# B&R Automation Studio project Panasonic_LinkaPowerCP2_A2021055 (part 24)

#### Main.st - Init, cyclic, exit code
```iecst
PROGRAM _INIT

END_PROGRAM

PROGRAM _CYCLIC

	//Volanie funkcie SequenceControl//
	SequenceControl(SC:= SC_P2_Cistenie);

	//Volanie podprogramov//
	OvlDveri;

	//Reset sekcie //
	IF P2_Cistenie.Reset THEN
		SC_P2_Cistenie.Step:= 0;
		P2_Cistenie.Reset:= FALSE;
	ELSIF NOT Safety.STAV.Linka_ZonaCS_AKTIVNA THEN
		SC_P2_Cistenie.Step:= 0;
	END_IF

	CASE SC_P2_Cistenie.Step OF

		0:
			SC_P2_Cistenie.StepName:='0 - Nulovanie';
			SC_OvlDveri.Step:= 0;
			P2_Cistenie.Automat:= FALSE;
			P2_Cistenie.KoniecCyklu:= FALSE;
			P2_Cistenie.Manual:= FALSE;
			P2_Cistenie.STAV.PoINIT:= FALSE;
			P2_Cistenie.OUT.Ionizator_OFF:= TRUE;
			P2_Cistenie.OUT.OdsavanieOfuk_ON:= FALSE;
			P2_Cistenie.OUT.Odsavanie_ON:= FALSE;
			P2_Cistenie.OUT.VzduchPreIonizator_ON:= FALSE;
			P2_Robot.COM_OUT.Cistenie_BezpecnaPozicia:= FALSE;
			P2_Robot.COM_OUT.Cistenie_OdoberPowerCP_4F:= FALSE;
			P2_Robot.COM_OUT.Cistenie_OdoberPowerCP_5F:= FALSE;
			P2_Robot.COM_OUT.Cistenie_OdoberPowerCP_5H:= FALSE;
			P2_Robot.COM_OUT.Cistenie_OtacajPowerCP:= FALSE;
			P2_Robot.COM_OUT.Cistenie_PolozPowerCP_4F:= FALSE;
			P2_Robot.COM_OUT.Cistenie_PolozPowerCP_5F:= FALSE;
			P2_Robot.COM_OUT.Cistenie_PolozPowerCP_5H:= FALSE;

			P2_Cistenie.COM_OUT.Stav_CistenieUkoncene:= FALSE;

			IF Safety.STAV.Linka_ZonaCS_AKTIVNA AND
				Safety.STAV.P2_ZonaBunky_AKTIVNA AND
				P2_Pracovisko.STAV.HardwareBunky_OK AND
				NOT P2_Pracovisko.STAV.Porucha_ST2 AND
				NOT P2_Pracovisko.STAV.Porucha_ST3 AND
				NOT P2_Pracovisko.STAV.Porucha_ST4 AND
				NOT P2_Pracovisko.STAV.Porucha_ST5 THEN
				SC_P2_Cistenie.ResetStep:= TRUE;
				SC_P2_Cistenie.Step:= 1;
			END_IF

		1:
			SC_P2_Cistenie.StepName:='1 - Cakam na spustenie vyroby';
			P2_Cistenie.KoniecCyklu:= FALSE;
			IF P2_Cistenie.Automat THEN
				SC_P2_Cistenie.Step:= 2;
			ELSIF P2_Cistenie.Manual THEN
				SC_P2_Cistenie.Step:= 700;
			END_IF

			//********************************************************Inicializácia****************************************************************************//

		2:
			SC_P2_Cistenie.StepName:='2 - Inicializacia - cakam na spustenie inicializacie';
			SC_P2_Cistenie.IdleTime.PT:= T#500ms;
			SC_P2_Cistenie.AlarmTime.PT:= T#5s;
			SC_P2_Cistenie.IdleTime.IN:= TRUE;

			IF SC_P2_Cistenie.IdleTime.Q THEN
				SC_P2_Cistenie.ResetStep:= TRUE;
				SC_P2_Cistenie.Step:= 3;
			END_IF

		3:
			SC_P2_Cistenie.StepName:='2 - Inicializacia - otvorenie dveri';
			SC_P2_Cistenie.IdleTime.PT:= T#500ms;
			SC_P2_Cistenie.AlarmTime.PT:= T#5s;

			IF NOT SC_P2_Cistenie.Switch1 THEN
				Dvere_OTVOR:= TRUE;
				SC_P2_Cistenie.Switch1:= TRUE;
			END_IF

			IF P2_Cistenie.IN.Dvere_OTVORENE THEN
				P2_Robot.COM_OUT.Cistenie_BezpecnaPozicia:= TRUE;
				P2_Cistenie.STAV.PoINIT:= TRUE;
				SC_P2_Cistenie.ResetStep:= TRUE;
				SC_P2_Cistenie.Step:= 100;
			END_IF

			//********************************************************Automatický režim****************************************************************************//

		100:
			SC_P2_Cistenie.StepName:='100 - Automaticky Rezim - cakam na spustenie cistenia';
			SC_P2_Cistenie.IdleTime.PT:= T#200ms;
			SC_P2_Cistenie.AlarmTime.PT:= T#5s;

			IF P2_Cistenie.KoniecCyklu AND NOT P2_StoperZvarania.Automat THEN
				SC_P2_Cistenie.ResetStep:= TRUE;
				SC_P2_Cistenie.Step:= 0;
			ELSIF P2_Cistenie.COM_IN.Cistenie_START THEN
				SC_P2_Cistenie.ResetStep:= TRUE;
				SC_P2_Cistenie.Step:= 102;
			END_IF

		102:
			SC_P2_Cistenie.StepName:='102 - Automaticky Rezim - vystavenie signalu pre robota odober Power CP z paletky a presun do cistenia';
			SC_P2_Cistenie.IdleTime.PT:= T#200ms;
			SC_P2_Cistenie.AlarmTime.PT:= T#5s;

			IF NOT P2_Robot.COM_IN.Stav_Cistenie_PowerCP_v_Cisteni AND NOT P2_Cistenie.IN.Vakum_OK THEN
				P2_Robot.COM_OUT.Cistenie_BezpecnaPozicia:= TRUE;
				IF Linka.PAR.ZvolenyModel = '4F' THEN
					P2_Robot.COM_OUT.Cistenie_OdoberPowerCP_4F:= TRUE;
					P2_Cistenie.OUT.Odsavanie_ON:= TRUE;
					SC_P2_Cistenie.ResetStep:= TRUE;
					SC_P2_Cistenie.Step:= 105;
				ELSIF Linka.PAR.ZvolenyModel = '5F' THEN
					P2_Robot.COM_OUT.Cistenie_OdoberPowerCP_5F:= TRUE;
					P2_Cistenie.OUT.Odsavanie_ON:= TRUE;
					SC_P2_Cistenie.ResetStep:= TRUE;
					SC_P2_Cistenie.Step:= 105;
				ELSIF Linka.PAR.ZvolenyModel = '5H' THEN
					P2_Robot.COM_OUT.Cistenie_OdoberPowerCP_5H:= TRUE;
					P2_Cistenie.OUT.Odsavanie_ON:= TRUE;
					SC_P2_Cistenie.ResetStep:= TRUE;
					SC_P2_Cistenie.Step:= 105;
				END_IF
			END_IF

		105:
			SC_P2_Cistenie.StepName:='105 - Automaticky Rezim - cakam na signal robot odobral Power CP z paletky';
			SC_P2_Cistenie.IdleTime.PT:= T#200ms;
			SC_P2_Cistenie.AlarmTime.PT:= T#5s;

			IF P2_Robot.COM_IN.Stav_Cistenie_PowerCP_v_Cisteni THEN
				P2_Robot.COM_OUT.Cistenie_OdoberPowerCP_4F:= FALSE;
				P2_Robot.COM_OUT.Cistenie_OdoberPowerCP_5F:= FALSE;
				P2_Robot.COM_OUT.Cistenie_OdoberPowerCP_5H:= FALSE;
				SC_P2_Cistenie.ResetStep:= TRUE;
				SC_P2_Cistenie.Step:= 108;
			END_IF

		108:
			SC_P2_Cistenie.StepName:='108 - Automaticky Rezim - zatvorenie dveri, spustenie ionizatora';
			SC_P2_Cistenie.IdleTime.PT:= T#2s;
			SC_P2_Cistenie.AlarmTime.PT:= T#5s;

			IF NOT SC_P2_Cistenie.Switch1 THEN
				P2_Cistenie.OUT.Ionizator_OFF:= FALSE;
				P2_Cistenie.OUT.VzduchPreIonizator_ON:= TRUE;
				Dvere_ZATVOR:= TRUE;
				P2_Robot.COM_OUT.Cistenie_BezpecnaPozicia:= FALSE;
				SC_P2_Cistenie.Switch1:= TRUE;
			END_IF

			IF P2_Cistenie.IN.Dvere_ZATVORENE THEN
				SC_P2_Cistenie.ResetStep:= TRUE;
				SC_P2_Cistenie.Step:= 112;
			END_IF

		112:
			SC_P2_Cistenie.StepName:='112 - Automaticky Rezim - zapnutie ofuku';
			SC_P2_Cistenie.IdleTime.PT:= T#2s;
			SC_P2_Cistenie.AlarmTime.PT:= T#5s;

			IF P2_Cistenie.IN.Vakum_OK THEN
				P2_Cistenie.OUT.OdsavanieOfuk_ON:= TRUE;
				SC_P2_Cistenie.ResetStep:= TRUE;
				SC_P2_Cistenie.Step:= 115;
			END_IF

		115:
			SC_P2_Cistenie.StepName:='115 - Automaticky Rezim - vystavenie signalu pre robota vykonaj otacanie Power CP v cisteni';
			SC_P2_Cistenie.IdleTime.PT:= T#200ms;
			SC_P2_Cistenie.AlarmTime.PT:= T#5s;

			IF NOT P2_Robot.COM_IN.Stav_Cistenie_Otacanie_Ukoncene THEN
				P2_Robot.COM_OUT.Cistenie_OtacajPowerCP:= TRUE;
				SC_P2_Cistenie.ResetStep:= TRUE;
				SC_P2_Cistenie.Step:= 118;
			END_IF

		118:
			SC_P2_Cistenie.StepName:='118 - Automaticky Rezim - cakam na signal robot ukoncil otacanie Power CP';
			SC_P2_Cistenie.IdleTime.PT:= T#200ms;
			SC_P2_Cistenie.AlarmTime.PT:= T#5s;

			IF P2_Robot.COM_IN.Stav_Cistenie_Otacanie_Ukoncene THEN
				P2_Robot.COM_OUT.Cistenie_OtacajPowerCP:= FALSE;
				SC_P2_Cistenie.ResetStep:= TRUE;
				SC_P2_Cistenie.Step:= 120;
			END_IF

		120:
			SC_P2_Cistenie.StepName:='120 - Automaticky Rezim - otvorenie dveri,vypnutie ofuku a odsavania';
			SC_P2_Cistenie.IdleTime.PT:= T#2s;
			SC_P2_Cistenie.AlarmTime.PT:= T#5s;

			IF NOT SC_P2_Cistenie.Switch1 THEN
				P2_Cistenie.OUT.OdsavanieOfuk_ON:= FALSE;
				P2_Cistenie.OUT.Odsavanie_ON:= FALSE;
				Dvere_OTVOR:= TRUE;
				SC_P2_Cistenie.Switch1:= TRUE;
			END_IF

			IF P2_Cistenie.IN.Dvere_OTVORENE THEN
				P2_Cistenie.OUT.Ionizator_OFF:= TRUE;
				P2_Cistenie.OUT.VzduchPreIonizator_ON:= FALSE;
				P2_Robot.COM_OUT.Cistenie_BezpecnaPozicia:= TRUE;
				SC_P2_Cistenie.ResetStep:= TRUE;
				SC_P2_Cistenie.Step:= 122;
			END_IF

		122:
			SC_P2_Cistenie.StepName:='122 - Automaticky Rezim - vystavenie signalu pre robota poloz Power CP na paletku po cisteni';
			SC_P2_Cistenie.IdleTime.PT:= T#200ms;
			SC_P2_Cistenie.AlarmTime.PT:= T#5s;

			IF NOT P2_Robot.COM_IN.Stav_Cistenie_PowerCP_Polozene THEN
				IF Linka.PAR.ZvolenyModel = '4F' THEN
					P2_Robot.COM_OUT.Cistenie_PolozPowerCP_4F:= TRUE;
					SC_P2_Cistenie.ResetStep:= TRUE;
					SC_P2_Cistenie.Step:= 125;
				ELSIF Linka.PAR.ZvolenyModel = '5F' THEN
					P2_Robot.COM_OUT.Cistenie_PolozPowerCP_5F:= TRUE;
					SC_P2_Cistenie.ResetStep:= TRUE;
					SC_P2_Cistenie.Step:= 125;
				ELSIF Linka.PAR.ZvolenyModel = '5H' THEN
					P2_Robot.COM_OUT.Cistenie_PolozPowerCP_5H:= TRUE;
					SC_P2_Cistenie.ResetStep:= TRUE;
					SC_P2_Cistenie.Step:= 125;
				END_IF
			END_IF

		125:
			SC_P2_Cistenie.StepName:='125 - Automaticky Rezim - cakam na signal robot polozil Power CP na paletku';
			SC_P2_Cistenie.IdleTime.PT:= T#200ms;
			SC_P2_Cistenie.AlarmTime.PT:= T#5s;

			IF P2_Robot.COM_IN.Stav_Cistenie_PowerCP_Polozene THEN
				P2_Robot.COM_OUT.Cistenie_PolozPowerCP_4F:= FALSE;
				P2_Robot.COM_OUT.Cistenie_PolozPowerCP_5F:= FALSE;
				P2_Robot.COM_OUT.Cistenie_PolozPowerCP_5H:= FALSE;
				SC_P2_Cistenie.ResetStep:= TRUE;
				SC_P2_Cistenie.Step:= 128;
			END_IF

		128:
			SC_P2_Cistenie.StepName:='122 - Automaticky Rezim - vystavenie signalu ukoncenie cistenia';
			SC_P2_Cistenie.IdleTime.PT:= T#200ms;
			SC_P2_Cistenie.AlarmTime.PT:= T#5s;

			IF NOT SC_P2_Cistenie.Switch1 THEN
				P2_Cistenie.COM_OUT.Stav_CistenieUkoncene:= TRUE;
				SC_P2_Cistenie.Switch1:= TRUE;
			END_IF

			IF NOT P2_Cistenie.COM_IN.Cistenie_START THEN
				P2_Cistenie.COM_OUT.Stav_CistenieUkoncene:= FALSE;
				SC_P2_Cistenie.ResetStep:= TRUE;
				SC_P2_Cistenie.Step:= 100;
			END_IF

			//**************************************************Ručný režim***********************************************************//

		700:
			SC_P2_Cistenie.StepName:='700 - Rucny rezim';
			SC_P2_Cistenie.IdleTime.PT:= T#200ms;
			SC_P2_Cistenie.AlarmTime.PT:= T#5s;

			//Otvorenie zatvorenie čistenia//
			IF P2_Cistenie.CMD.RR_Cistenie_OTVOR THEN
				Dvere_OTVOR:= TRUE;
				P2_Cistenie.CMD.RR_Cistenie_OTVOR:= FALSE;
			ELSIF P2_Cistenie.CMD.RR_Cistenie_ZATVOR THEN
				Dvere_ZATVOR:= TRUE;
				P2_Cistenie.CMD.RR_Cistenie_ZATVOR:= FALSE;
			END_IF

	END_CASE

END_PROGRAM

PROGRAM _EXIT
	(* Insert code here *)

END_PROGRAM
```

#### Variables.var - Local variables
```iecst
VAR
	SC_OvlDveri : SequenceControlTyp;
	Dvere_OTVOR : BOOL;
	Dvere_ZATVOR : BOOL;
END_VAR
```

#### OvlDveri.st
```iecst
ACTION OvlDveri:

	//Volanie funkcie SequenceControl//
	SequenceControl(SC:= SC_OvlDveri);

	CASE SC_OvlDveri.Step OF

		0:
			SC_OvlDveri.StepName:= '0 - Nulovanie';
			Dvere_OTVOR:= FALSE;
			Dvere_ZATVOR:= FALSE;
			P2_Cistenie.OUT.Dvere_OTVOR:= FALSE;
			P2_Cistenie.OUT.Dvere_ZATVOR:= FALSE;

			IF SC_P2_Cistenie.Step <> 0 THEN
				SC_OvlDveri.ResetStep:= TRUE;
				SC_OvlDveri.Step:= 1;
			END_IF

		1:
			SC_OvlDveri.StepName:= '1 - Rozhodnutie o cinnosti';
			IF Dvere_OTVOR THEN
				SC_OvlDveri.Step:= 10;
			ELSIF Dvere_ZATVOR THEN
				SC_OvlDveri.Step:= 20;
			END_IF

		10:
			SC_OvlDveri.StepName:= '10 - Otvorenie dveri';
			SC_OvlDveri.IdleTime.PT:= T#3s;
			SC_OvlDveri.AlarmTime.PT:= T#3s;

			IF P2_Cistenie.Automat THEN
				SC_OvlDveri.AlarmTime.IN:= TRUE;
			ELSE
				SC_OvlDveri.IdleTime.IN:= TRUE;
			END_IF

			IF NOT SC_OvlDveri.Switch1 THEN
				P2_Cistenie.OUT.Dvere_OTVOR:= TRUE;
				SC_OvlDveri.Switch1:= TRUE;
			END_IF

			IF P2_Cistenie.IN.Dvere_OTVORENE OR SC_OvlDveri.IdleTime.Q THEN
				SC_OvlDveri.ResetStep:= TRUE;
				SC_OvlDveri.Step:= 0;
			ELSIF SC_OvlDveri.AlarmTime.Q THEN
				P2_Alarmy[224]:= TRUE;
				P2_Pracovisko.STAV.Porucha_ST5:= TRUE;
			END_IF

		20:
			SC_OvlDveri.StepName:= '20 - Zatvorenie dveri';
			SC_OvlDveri.IdleTime.PT:= T#3s;
			SC_OvlDveri.AlarmTime.PT:= T#3s;

			IF P2_Cistenie.Automat THEN
				SC_OvlDveri.AlarmTime.IN:= TRUE;
			ELSE
				SC_OvlDveri.IdleTime.IN:= TRUE;
			END_IF

			IF NOT SC_OvlDveri.Switch1 THEN
				P2_Cistenie.OUT.Dvere_ZATVOR:= TRUE;
				SC_OvlDveri.Switch1:= TRUE;
			END_IF

			IF P2_Cistenie.IN.Dvere_ZATVORENE OR SC_OvlDveri.IdleTime.Q THEN
				SC_OvlDveri.ResetStep:= TRUE;
				SC_OvlDveri.Step:= 0;
			ELSIF SC_OvlDveri.AlarmTime.Q THEN
				P2_Alarmy[223]:= TRUE;
				P2_Pracovisko.STAV.Porucha_ST5:= TRUE;
			END_IF

	END_CASE

END_ACTION
```

### Program Logical/Program/Pracovisko_2/P2_OvladVizu (IEC)

#### Main.st - Init, cyclic, exit code
```iecst
PROGRAM _INIT
	(* Insert code here *)

END_PROGRAM

PROGRAM _CYCLIC

	//*************************************Prepnutie obrazovky pri stlačení tlačítka CS*********************************//
	IF EDGEPOS(P2_Pracovisko.STAV.Manual AND NOT Safety.STAV.Linka_ZonaCS_AKTIVNA) THEN
		P2_Vizu.GoPage:= 'PageAutomatP2';
	END_IF

	//************************************Filter alarmov**************************************************************//
	FilterVizu_P2:= '[{"logicalOperator":"and","value":200,"conditionType":">=","columnType":"cod","useAlarmState":false,"alarmState":0},{"value":299,"conditionType":"<=","columnType":"cod","useAlarmState":false,"alarmState":0}]';

	//**********************************Zobrazenie upozornenia na kontrolu skrutiek na stanici 5 skrutkovania***********************************//
	IF EDGEPOS(Linka.PAR.ZvolenyModel = '4F')THEN
		P2_Vizu.ZobrazHL5_ST5:= TRUE;
		P2_Vizu.ZobrazHL6_ST5:= FALSE;
		P2_Vizu.ZobrazHL7_ST5:= FALSE;
	END_IF

	IF EDGEPOS(Linka.PAR.ZvolenyModel = '5F')THEN
		P2_Vizu.ZobrazHL5_ST5:= FALSE;
		P2_Vizu.ZobrazHL6_ST5:= TRUE;
		P2_Vizu.ZobrazHL7_ST5:= FALSE;
	END_IF

	IF EDGEPOS(Linka.PAR.ZvolenyModel = '5H')THEN
		P2_Vizu.ZobrazHL5_ST5:= FALSE;
		P2_Vizu.ZobrazHL6_ST5:= FALSE;
		P2_Vizu.ZobrazHL7_ST5:= TRUE;
	END_IF

	//Zmeny farieb tlačítok ovládania zámkov//
	//Zadné dvere //
	IF P2_Pracovisko.STAV.ZadneDvereZamknute AND P2_Pracovisko.IN.ZadneDvereLS_PritomnostAdaptera AND P2_Pracovisko.IN.ZadneDverePS_PritomnostAdaptera THEN
		P2_Vizu.TL_ZadnyZamok_Farba:= "Button_Green";
	ELSIF P2_Pracovisko.IN.ZadneDvereLS_PritomnostAdaptera AND P2_Pracovisko.IN.ZadneDverePS_PritomnostAdaptera THEN
		IF Blikac1s THEN
			P2_Vizu.TL_ZadnyZamok_Farba:= "Button_Blue";
		ELSE
			P2_Vizu.TL_ZadnyZamok_Farba:= "Operate";
		END_IF
	ELSE
		P2_Vizu.TL_ZadnyZamok_Farba:= "Button_Red";
	END_IF

	//Predné dvere //
	IF P2_Pracovisko.STAV.PredneDvereZamknute AND P2_Pracovisko.IN.PredneDvereLS_PritomnostAdaptera AND P2_Pracovisko.IN.PredneDverePS_PritomnostAdaptera THEN
		P2_Vizu.TL_PrednyZamok_Farba:= "Button_Green";
	ELSIF P2_Pracovisko.IN.PredneDvereLS_PritomnostAdaptera AND P2_Pracovisko.IN.PredneDverePS_PritomnostAdaptera THEN
		IF Blikac1s THEN
			P2_Vizu.TL_PrednyZamok_Farba:= "Button_Blue";
		ELSE
			P2_Vizu.TL_PrednyZamok_Farba:= "Operate";
		END_IF
	ELSE
		P2_Vizu.TL_PrednyZamok_Farba:= "Button_Red";
	END_IF

	//***********************************Zobrazenie warningov pracoviska****************************************************//
	//0 - Pracovisko je vypnuté.
	//1 - Prebieha inicializácia pracoviska.
	//2 - Na pracovisku prebieha výroba.
	//3 - Prebieha ukončenie pracovného cyklu pracoviska.
	//4 - Prebieha režim vyprázdnenia linky.
	//5 - Robot nie je prepnuty do automatického režimu !!!
	//6 - Doplň zásobník matíc M4 !!!
	//7 - Doplň zásobník skrutiek M4 !!!
	//8 - Doplň zásobník skrutiek M5 !!!
	//9 - Doplň zásobník skrutiek M6 !!!

	IF NOT P2_Robot.COM_IN.Stav_RezimAUTOMAT THEN
		P2_Vizu.Warnings_Index:= 5;
	ELSIF P2_Pracovisko.STAV.Automat AND NOT P2_Pracovisko.STAV.PoINIT AND NOT P2_Pracovisko.STAV.UkoncenieCyklu_BUSY THEN
		P2_Vizu.Warnings_Index:= 1;
	ELSIF P2_StoperMaticovacky.SkrutSet_MaticaM4.IN.ZasobnikMaticPrazdny THEN
		P2_Vizu.Warnings_Index:= 6;
	ELSIF P2_Srobovanie.SkrutSet_M4.IN.ZasobnikSkrutiekPrazdny THEN
		P2_Vizu.Warnings_Index:= 7;
	ELSIF P2_Srobovanie.SkrutSet_M5.IN.VibracnyHrniec.PritomnostSkrutiekVHrnci THEN
		P2_Vizu.Warnings_Index:= 8;
	ELSIF P2_Srobovanie.SkrutSet_M6.IN.VibracnyHrniec.PritomnostSkrutiekVHrnci THEN
		P2_Vizu.Warnings_Index:= 9;
	ELSIF Linka.PAR.TestovaciKus THEN
		P2_Vizu.Warnings_Index:= 11;
	ELSIF Linka.PAR.VyprazdnenieLinky THEN
		P2_Vizu.Warnings_Index:= 4;
	ELSIF P2_Pracovisko.STAV.PoINIT AND NOT P2_Pracovisko.STAV.UkoncenieCyklu_BUSY THEN
		P2_Vizu.Warnings_Index:= 2;
	ELSIF P2_Pracovisko.STAV.UkoncenieCyklu_BUSY THEN
		P2_Vizu.Warnings_Index:= 3;
	ELSIF NOT P2_Pracovisko.STAV.Automat THEN
		P2_Vizu.Warnings_Index:= 0;
	END_IF

	//************************Prepínanie farby textového pola warning zariadenia***********************************//
	IF P2_Vizu.Warnings_Index = 0 THEN
		P2_Vizu.Warnings_Farba:= "TextOutput_Grey";
	ELSIF P2_Vizu.Warnings_Index = 1 THEN
		P2_Vizu.Warnings_Farba:= "TextOutput_Blue";
	ELSIF P2_Vizu.Warnings_Index = 2 THEN
		P2_Vizu.Warnings_Farba:= "TextOutput_Green";
	ELSIF P2_Vizu.Warnings_Index = 3 THEN
		P2_Vizu.Warnings_Farba:= "TextOutput_Blue";
	ELSIF P2_Vizu.Warnings_Index = 4 THEN
		P2_Vizu.Warnings_Farba:= "TextOutput_Green";
	ELSIF P2_Vizu.Warnings_Index = 11 THEN
		P2_Vizu.Warnings_Farba:= "TextOutput_Green";
	ELSE
		IF Blikac1s THEN
			P2_Vizu.Warnings_Farba:= "TextOutput_Orange";
		ELSE
			P2_Vizu.Warnings_Farba:= "TextOutput_Grey";
		END_IF
	END_IF

	//***********************Prepnutie bootovacej obrazovky********************************//
	IF P2_Vizu.ActualPage <> 'PageBootP2' AND NOT Safety.STAV.Linka_SafetyPLC_Nabehlo THEN
		P2_Vizu.GoPage:= 'PageBootP2';
	ELSIF P2_Vizu.ActualPage = 'PageBootP2' AND Safety.STAV.Linka_SafetyPLC_Nabehlo THEN
		P2_Vizu.GoPage:= 'PageAutomatP2';
	END_IF

	IF P2_Vizu.GoPage = 'PageBootP2' AND P2_Vizu.ActualPage = 'PageBootP2' THEN
		P2_Vizu.GoPage:= '';
	ELSIF P2_Vizu.GoPage = 'PageAutomatP2' AND P2_Vizu.ActualPage = 'PageAutomatP2' THEN
		P2_Vizu.GoPage:= '';
	END_IF

	//********************************Blikanie tlačítka Alarmy*******************************************************//
	IF P2_Pracovisko.STAV.PORUCHA AND P2_Vizu.ActualPage <> 'PageAlarmP2' THEN
		IF Blikac500ms THEN
			P2_AlarmyVizu.FarbaTlacitka_Alarmy:= "Button_Red";
		ELSE
			P2_AlarmyVizu.FarbaTlacitka_Alarmy:= "default";
		END_IF
	ELSE
		P2_AlarmyVizu.FarbaTlacitka_Alarmy:= "default";
	END_IF

	//*************************************Zamknutie tlačítok***************************************************************//
	//Zamknutie tlačítok ovládania zámkov//
	IF P2_Pracovisko.STAV.Automat THEN
		P2_Vizu.TL_OvladaniaZamkov_ENABLE:= FALSE;
	ELSIF P2_Srobovanie.STAV.RR_Polohovanie_BUSY THEN
		P2_Vizu.TL_OvladaniaZamkov_ENABLE:= FALSE;
	ELSIF P2_Srobovanie.STAV.CistenieSkrutkovackyM5_BUSY THEN
		P2_Vizu.TL_OvladaniaZamkov_ENABLE:= FALSE;
	ELSIF P2_Srobovanie.STAV.CistenieSkrutkovackyM6_BUSY THEN
		P2_Vizu.TL_OvladaniaZamkov_ENABLE:= FALSE;
	ELSIF P2_Zvaranie.STAV.RR_SekvenciaZvarania_BUSY THEN
		P2_Vizu.TL_OvladaniaZamkov_ENABLE:= FALSE;
	ELSE
		P2_Vizu.TL_OvladaniaZamkov_ENABLE:= TRUE;
	END_IF

	//Tlačítko Štat Automat//
	IF P2_Pracovisko.STAV.UkoncenieCyklu_BUSY THEN
		P2_Vizu.TL_StartAutomat_ENABLE:= FALSE;
	ELSIF P2_Pracovisko.STAV.PORUCHA THEN
		P2_Vizu.TL_StartAutomat_ENABLE:= FALSE;
	ELSIF NOT P2_Robot.COM_IN.Stav_RezimAUTOMAT THEN
		P2_Vizu.TL_StartAutomat_ENABLE:= FALSE;
	ELSIF NOT Safety.STAV.P2_ZonaBunky_AKTIVNA THEN
		P2_Vizu.TL_StartAutomat_ENABLE:= FALSE;
	ELSIF NOT P2_Pracovisko.STAV.HardwareZaklTesnenia_OK THEN
		P2_Vizu.TL_StartAutomat_ENABLE:= FALSE;
	ELSIF NOT P2_Pracovisko.STAV.HardwareBunky_OK THEN
		P2_Vizu.TL_StartAutomat_ENABLE:= FALSE;
	ELSE
		P2_Vizu.TL_StartAutomat_ENABLE:= TRUE;
	END_IF

	//Tlačítko Ukončenie Cyklu//
	IF P2_Pracovisko.STAV.PoINIT THEN
		P2_Vizu.TL_KoniecCyklu_ENABLE:= TRUE;
	ELSE
		P2_Vizu.TL_KoniecCyklu_ENABLE:= FALSE;
	END_IF

	//Tlačítko STOP//
	IF P2_Pracovisko.STAV.PoINIT AND NOT P2_Pracovisko.STAV.UkoncenieCyklu_BUSY THEN
		P2_Vizu.TL_STOP_ENABLE:= FALSE;
	ELSE
		P2_Vizu.TL_STOP_ENABLE:= TRUE;
	END_IF

	//Tlačítko Režim Automat//
	P2_Vizu.TL_RezimAutomat_ENABLE:= TRUE;

	//Tlačítko Režim Manual//
	IF P2_Pracovisko.STAV.Automat THEN
		P2_Vizu.TL_RezimManual_ENABLE:= FALSE;
	ELSIF NOT P2_Pracovisko.STAV.HardwareZaklTesnenia_OK THEN
		P2_Vizu.TL_RezimManual_ENABLE:= FALSE;
	ELSIF NOT P2_Pracovisko.STAV.HardwareBunky_OK THEN
		P2_Vizu.TL_RezimManual_ENABLE:= FALSE;
	ELSE
		P2_Vizu.TL_RezimManual_ENABLE:= TRUE;
	END_IF

	//RR - Tlačítko vysunutia maticovačky//
	IF NOT Safety.STAV.P2_ZonaBunky_AKTIVNA THEN
		P2_Vizu.TL_VysunutiaMaticovacM4_ENABLE:= FALSE;
	ELSE
		P2_Vizu.TL_VysunutiaMaticovacM4_ENABLE:= TRUE;
	END_IF

	//RR - Tlačítko čistenia skrutkovačky M6//
	IF P2_Srobovanie.STAV.RR_Polohovanie_BUSY THEN
		P2_Vizu.TL_VycistiSkrutkovackuM6_ENABLE:= FALSE;
	ELSIF NOT Safety.STAV.P2_ZonaBunky_AKTIVNA THEN
		P2_Vizu.TL_VycistiSkrutkovackuM6_ENABLE:= FALSE;
	ELSIF NOT Safety.STAV.Linka_ZonaCS_AKTIVNA THEN
		P2_Vizu.TL_VycistiSkrutkovackuM6_ENABLE:= FALSE;
	ELSIF P2_Srobovanie.STAV.CistenieSkrutkovackyM6_BUSY THEN
		P2_Vizu.TL_VycistiSkrutkovackuM6_ENABLE:= FALSE;
	ELSIF P2_Srobovanie.STAV.CistenieSkrutkovackyM5_BUSY THEN
		P2_Vizu.TL_VycistiSkrutkovackuM6_ENABLE:= FALSE;
	ELSIF NOT P2_Pracovisko.STAV.SkrutkovackyZasunute THEN
		P2_Vizu.TL_VycistiSkrutkovackuM6_ENABLE:= FALSE;
	ELSIF P2_Srobovanie.CMD.RR_SkrutSetM6_VysunBrzdu THEN
		P2_Vizu.TL_VycistiSkrutkovackuM6_ENABLE:= FALSE;
	ELSIF P2_Srobovanie.CMD.RR_SkrutSetM6_Zasobnik_RUN THEN
		P2_Vizu.TL_VycistiSkrutkovackuM6_ENABLE:= FALSE;
	ELSE
		P2_Vizu.TL_VycistiSkrutkovackuM6_ENABLE:= TRUE;
	END_IF

	//RR - Tlačítko čistenia skrutkovačky M5//
	IF P2_Srobovanie.STAV.RR_Polohovanie_BUSY THEN
		P2_Vizu.TL_VycistiSkrutkovackuM5_ENABLE:= FALSE;
	ELSIF NOT Safety.STAV.P2_ZonaBunky_AKTIVNA THEN
		P2_Vizu.TL_VycistiSkrutkovackuM5_ENABLE:= FALSE;
	ELSIF NOT Safety.STAV.Linka_ZonaCS_AKTIVNA THEN
		P2_Vizu.TL_VycistiSkrutkovackuM5_ENABLE:= FALSE;
	ELSIF P2_Srobovanie.STAV.CistenieSkrutkovackyM6_BUSY THEN
		P2_Vizu.TL_VycistiSkrutkovackuM5_ENABLE:= FALSE;
	ELSIF P2_Srobovanie.STAV.CistenieSkrutkovackyM5_BUSY THEN
		P2_Vizu.TL_VycistiSkrutkovackuM5_ENABLE:= FALSE;
	ELSIF NOT P2_Pracovisko.STAV.SkrutkovackyZasunute THEN
		P2_Vizu.TL_VycistiSkrutkovackuM5_ENABLE:= FALSE;
	ELSIF P2_Srobovanie.CMD.RR_SkrutSetM5_VysunBrzdu THEN
		P2_Vizu.TL_VycistiSkrutkovackuM5_ENABLE:= FALSE;
	ELSIF P2_Srobovanie.CMD.RR_SkrutSetM5_Zasobnik_RUN THEN
		P2_Vizu.TL_VycistiSkrutkovackuM5_ENABLE:= FALSE;
	ELSE
		P2_Vizu.TL_VycistiSkrutkovackuM5_ENABLE:= TRUE;
	END_IF

	//RR - Tlačítko polohovania aplikátora//
	IF P2_Srobovanie.STAV.RR_Polohovanie_BUSY THEN
		P2_Vizu.TL_PolohujManipulator_ENABLE:= FALSE;
	ELSIF NOT Safety.STAV.P2_ZonaBunky_AKTIVNA THEN
		P2_Vizu.TL_PolohujManipulator_ENABLE:= FALSE;
	ELSIF NOT Safety.STAV.Linka_ZonaCS_AKTIVNA THEN
		P2_Vizu.TL_PolohujManipulator_ENABLE:= FALSE;
	ELSIF P2_Srobovanie.STAV.CistenieSkrutkovackyM6_BUSY THEN
		P2_Vizu.TL_PolohujManipulator_ENABLE:= FALSE;
	ELSIF P2_Srobovanie.STAV.CistenieSkrutkovackyM5_BUSY THEN
		P2_Vizu.TL_PolohujManipulator_ENABLE:= FALSE;
	ELSIF NOT P2_Pracovisko.STAV.SkrutkovackyZasunute THEN
		P2_Vizu.TL_PolohujManipulator_ENABLE:= FALSE;
	ELSE
		P2_Vizu.TL_PolohujManipulator_ENABLE:= TRUE;
	END_IF

	//RR - Tlačítko vysunutia skrutkovačky M6//
	IF P2_Srobovanie.STAV.RR_Polohovanie_BUSY THEN
		P2_Vizu.Tl_VysunutieSkrutkovM6_ENABLE:= FALSE;
	ELSIF P2_Srobovanie.STAV.CistenieSkrutkovackyM6_BUSY THEN
		P2_Vizu.Tl_VysunutieSkrutkovM6_ENABLE:= FALSE;
	ELSIF P2_Srobovanie.STAV.CistenieSkrutkovackyM5_BUSY THEN
		P2_Vizu.Tl_VysunutieSkrutkovM6_ENABLE:= FALSE;
	ELSIF NOT Safety.STAV.P2_ZonaBunky_AKTIVNA THEN
		P2_Vizu.Tl_VysunutieSkrutkovM6_ENABLE:= FALSE;
	ELSIF NOT Safety.STAV.Linka_ZonaCS_AKTIVNA THEN
		P2_Vizu.Tl_VysunutieSkrutkovM6_ENABLE:= FALSE;
	ELSE
		P2_Vizu.Tl_VysunutieSkrutkovM6_ENABLE:= TRUE;
	END_IF

	//RR - Tlačítko vysunutia skrutkovačky M5//
	IF P2_Srobovanie.STAV.RR_Polohovanie_BUSY THEN
		P2_Vizu.Tl_VysunutieSkrutkovM5_ENABLE:= FALSE;
	ELSIF P2_Srobovanie.STAV.CistenieSkrutkovackyM6_BUSY THEN
		P2_Vizu.Tl_VysunutieSkrutkovM5_ENABLE:= FALSE;
	ELSIF P2_Srobovanie.STAV.CistenieSkrutkovackyM5_BUSY THEN
		P2_Vizu.Tl_VysunutieSkrutkovM5_ENABLE:= FALSE;
	ELSIF NOT Safety.STAV.P2_ZonaBunky_AKTIVNA THEN
		P2_Vizu.Tl_VysunutieSkrutkovM5_ENABLE:= FALSE;
	ELSIF NOT Safety.STAV.Linka_ZonaCS_AKTIVNA THEN
		P2_Vizu.Tl_VysunutieSkrutkovM5_ENABLE:= FALSE;
	ELSE
		P2_Vizu.Tl_VysunutieSkrutkovM5_ENABLE:= TRUE;
	END_IF

	//RR - Tlačítko vysunutia skrutkovačky M4//
	IF P2_Srobovanie.STAV.RR_Polohovanie_BUSY THEN
		P2_Vizu.TL_OvladaniaVysunSkrutkovM4:= FALSE;
	ELSIF P2_Srobovanie.STAV.CistenieSkrutkovackyM6_BUSY THEN
		P2_Vizu.TL_OvladaniaVysunSkrutkovM4:= FALSE;
	ELSIF P2_Srobovanie.STAV.CistenieSkrutkovackyM5_BUSY THEN
		P2_Vizu.TL_OvladaniaVysunSkrutkovM4:= FALSE;
	ELSIF NOT Safety.STAV.P2_ZonaBunky_AKTIVNA THEN
		P2_Vizu.TL_OvladaniaVysunSkrutkovM4:= FALSE;
	ELSIF NOT Safety.STAV.Linka_ZonaCS_AKTIVNA THEN
		P2_Vizu.TL_OvladaniaVysunSkrutkovM4:= FALSE;
	ELSE
		P2_Vizu.TL_OvladaniaVysunSkrutkovM4:= TRUE;
	END_IF

	//RR - Ovládanie skrutkovacieho setu M6//
	IF P2_Srobovanie.STAV.CistenieSkrutkovackyM6_BUSY THEN
		P2_Vizu.TL_OvladSkrutkovSetuM6_ENABLE:= FALSE;
	ELSE
		P2_Vizu.TL_OvladSkrutkovSetuM6_ENABLE:= TRUE;
	END_IF

	//RR - Ovládanie skrutkovacieho setu M5//
	IF P2_Srobovanie.STAV.CistenieSkrutkovackyM5_BUSY THEN
		P2_Vizu.TL_OvladSkrutkovSetuM5_ENABLE:= FALSE;
	ELSE
		P2_Vizu.TL_OvladSkrutkovSetuM5_ENABLE:= TRUE;
	END_IF

	//RR - Ovládanie manipulatora XY//
	IF NOT Safety.STAV.P2_ZonaBunky_AKTIVNA THEN
		P2_Vizu.TL_OvladManipulatoraXY_ENABLE:= FALSE;
	ELSE
		P2_Vizu.TL_OvladManipulatoraXY_ENABLE:= TRUE;
	END_IF

	//RR - Ovládanie presunu zvárania//
	IF P2_Zvaranie.STAV.RR_SekvenciaZvarania_BUSY THEN
		P2_Vizu.TL_PresunZvarania_ENABLE:= FALSE;
	ELSIF P2_Zvaranie.ServoZdvihuZvarania.Status.ActPosition > 200 THEN
		P2_Vizu.TL_PresunZvarania_ENABLE:= FALSE;
	ELSE
		P2_Vizu.TL_PresunZvarania_ENABLE:= TRUE;
	END_IF

	//RR - Spustenie sekvencie zvárania//
	IF NOT Safety.STAV.P2_ZonaBunky_AKTIVNA THEN
		P2_Vizu.TL_StartSekvencieZvarania_ENABLE:= FALSE;
	ELSIF NOT Safety.STAV.Linka_ZonaCS_AKTIVNA THEN
		P2_Vizu.TL_StartSekvencieZvarania_ENABLE:= FALSE;
	ELSE
		P2_Vizu.TL_StartSekvencieZvarania_ENABLE:= TRUE;
	END_IF

	//RR - Ovládanie zdvihu zvárania//
	IF NOT Safety.STAV.P2_ZonaBunky_AKTIVNA THEN
		P2_Vizu.TL_ZdvihZvarania_ENABLE:= FALSE;
	ELSIF NOT P2_StoperZvarania.RFID_hlava.PritomnostPaletky THEN
		P2_Vizu.TL_ZdvihZvarania_ENABLE:= FALSE;
	ELSE
		P2_Vizu.TL_ZdvihZvarania_ENABLE:= TRUE;
	END_IF

	//**************************Zamknutie editácie parametrov*********************************//
	IF P2_UrovenPrihlasenehoUzivatela >= 20 THEN
		P2_Vizu.EditaciaParametrov_ENABLE:= TRUE;
	ELSE
		P2_Vizu.EditaciaParametrov_ENABLE:= FALSE;
	END_IF

	//***********************************Prepínanie stavov pracovísk*******************************************************************//
	//Dopravníky//
	IF P2_Dopravniky.Automat AND NOT P2_Dopravniky.STAV.PoINIT THEN
		P2_Vizu.IndexStavu_Dopravnik:= 1;
	ELSIF P2_Dopravniky.Automat AND P2_Dopravniky.STAV.PoINIT THEN
		P2_Vizu.IndexStavu_Dopravnik:= 2;
	ELSE
		P2_Vizu.IndexStavu_Dopravnik:= 0;
	END_IF

	//Stoper zakladania tesnenia//
	IF NOT P2_Pracovisko.STAV.HardwareZaklTesnenia_OK THEN
		P2_Vizu.IndexStavu_StoperZakladacaTesn:= 3;
	ELSIF P2_Pracovisko.STAV.Porucha_ST1 THEN
		P2_Vizu.IndexStavu_StoperZakladacaTesn:= 3;
	ELSIF P2_StoperZaklTesnenia.Automat AND NOT P2_StoperZaklTesnenia.STAV.PoINIT THEN
		P2_Vizu.IndexStavu_StoperZakladacaTesn:= 1;
	ELSIF P2_StoperZaklTesnenia.Automat AND P2_StoperZaklTesnenia.STAV.PoINIT THEN
		P2_Vizu.IndexStavu_StoperZakladacaTesn:= 2;
	ELSE
		P2_Vizu.IndexStavu_StoperZakladacaTesn:= 0;
	END_IF

	//Zakladač tesnenia//
	IF NOT P2_Pracovisko.STAV.HardwareZaklTesnenia_OK THEN
		P2_Vizu.IndexStavu_ZakladacaTesnenia:= 3;
	ELSIF P2_Pracovisko.STAV.Porucha_ST1 THEN
		P2_Vizu.IndexStavu_ZakladacaTesnenia:= 3;
	ELSIF P2_ZakladacTesnenia.Automat AND NOT P2_ZakladacTesnenia.STAV.PoINIT THEN
		P2_Vizu.IndexStavu_ZakladacaTesnenia:= 1;
	ELSIF P2_ZakladacTesnenia.Automat AND P2_ZakladacTesnenia.STAV.PoINIT THEN
		P2_Vizu.IndexStavu_ZakladacaTesnenia:= 2;
	ELSE
		P2_Vizu.IndexStavu_ZakladacaTesnenia:= 0;
	END_IF

	//Stoper maticovačky//
	IF NOT P2_Pracovisko.STAV.HardwareBunky_OK THEN
		P2_Vizu.IndexStavu_StoperMaticovacky:= 3;
	ELSIF P2_Pracovisko.STAV.Porucha_ST2 THEN
		P2_Vizu.IndexStavu_StoperMaticovacky:= 3;
	ELSIF P2_StoperMaticovacky.Automat AND NOT P2_StoperMaticovacky.STAV.PoINIT THEN
		P2_Vizu.IndexStavu_StoperMaticovacky:= 1;
	ELSIF P2_StoperMaticovacky.Automat AND P2_StoperMaticovacky.STAV.PoINIT THEN
		P2_Vizu.IndexStavu_StoperMaticovacky:= 2;
	ELSE
		P2_Vizu.IndexStavu_StoperMaticovacky:= 0;
	END_IF

	//Akumulačný stoper//
	IF P2_Pracovisko.STAV.Porucha_ST3 THEN
		P2_Vizu.IndexStavu_AkumulacnyStoper:= 3;
	ELSIF P2_AkumulacnyStoper.Automat AND NOT P2_AkumulacnyStoper.STAV.PoINIT THEN
		P2_Vizu.IndexStavu_AkumulacnyStoper:= 1;
	ELSIF P2_AkumulacnyStoper.Automat AND P2_AkumulacnyStoper.STAV.PoINIT THEN
		P2_Vizu.IndexStavu_AkumulacnyStoper:= 2;
	ELSE
		P2_Vizu.IndexStavu_AkumulacnyStoper:= 0;
	END_IF

	//Stoper šrobovania//
	IF NOT P2_Pracovisko.STAV.HardwareBunky_OK THEN
		P2_Vizu.IndexStavu_StoperSrobovania:= 3;
	ELSIF P2_Pracovisko.STAV.Porucha_ST4 THEN
		P2_Vizu.IndexStavu_StoperSrobovania:= 3;
	ELSIF P2_StoperSrobovania.Automat AND NOT P2_StoperSrobovania.STAV.PoINIT THEN
		P2_Vizu.IndexStavu_StoperSrobovania:= 1;
	ELSIF P2_StoperSrobovania.Automat AND P2_StoperSrobovania.STAV.PoINIT THEN
		P2_Vizu.IndexStavu_StoperSrobovania:= 2;
	ELSE
		P2_Vizu.IndexStavu_StoperSrobovania:= 0;
	END_IF

	//Šrobovanie//
	IF NOT P2_Pracovisko.STAV.HardwareBunky_OK THEN
		P2_Vizu.IndexStavu_Srobovania:= 3;
	ELSIF P2_Pracovisko.STAV.Porucha_ST4 THEN
		P2_Vizu.IndexStavu_Srobovania:= 3;
	ELSIF P2_Srobovanie.Automat AND NOT P2_Srobovanie.STAV.PoINIT THEN
		P2_Vizu.IndexStavu_Srobovania:= 1;
	ELSIF P2_Srobovanie.Automat AND P2_Srobovanie.STAV.PoINIT THEN
		P2_Vizu.IndexStavu_Srobovania:= 2;
	ELSE
		P2_Vizu.IndexStavu_Srobovania:= 0;
	END_IF

	//Robot//
	IF P2_Robot.Automat AND NOT P2_Robot.STAV.PoINIT THEN
		P2_Vizu.IndexStavu_Robot:= 1;
	ELSIF P2_Robot.Automat AND P2_Robot.STAV.PoINIT THEN
		P2_Vizu.IndexStavu_Robot:= 2;
	ELSE
		P2_Vizu.IndexStavu_Robot:= 0;
	END_IF

	//Stoper zvárania//
	IF NOT P2_Pracovisko.STAV.HardwareBunky_OK THEN
		P2_Vizu.IndexStavu_StoperZvarania:= 3;
	ELSIF P2_Pracovisko.STAV.Porucha_ST5 THEN
		P2_Vizu.IndexStavu_StoperZvarania:= 3;
	ELSIF P2_StoperZvarania.Automat AND NOT P2_StoperZvarania.STAV.PoINIT THEN
		P2_Vizu.IndexStavu_StoperZvarania:= 1;
	ELSIF P2_StoperZvarania.Automat AND P2_StoperZvarania.STAV.PoINIT THEN
		P2_Vizu.IndexStavu_StoperZvarania:= 2;
	ELSE
		P2_Vizu.IndexStavu_StoperZvarania:= 0;
	END_IF

	//Zváranie//
	IF NOT P2_Pracovisko.STAV.HardwareBunky_OK THEN
		P2_Vizu.IndexStavu_Zvaranie:= 3;
	ELSIF P2_Pracovisko.STAV.Porucha_ST5 THEN
		P2_Vizu.IndexStavu_Zvaranie:= 3;
	ELSIF P2_Zvaranie.Automat AND NOT P2_Zvaranie.STAV.PoINIT THEN
		P2_Vizu.IndexStavu_Zvaranie:= 1;
	ELSIF P2_Zvaranie.Automat AND P2_Zvaranie.STAV.PoINIT THEN
		P2_Vizu.IndexStavu_Zvaranie:= 2;
	ELSE
		P2_Vizu.IndexStavu_Zvaranie:= 0;
	END_IF

	//Čistenie//
	IF NOT P2_Pracovisko.STAV.HardwareBunky_OK THEN
		P2_Vizu.IndexStavu_Cistenie:= 3;
	ELSIF P2_Pracovisko.STAV.Porucha_ST5 THEN
		P2_Vizu.IndexStavu_Cistenie:= 3;
	ELSIF P2_Cistenie.Automat AND NOT P2_Cistenie.STAV.PoINIT THEN
		P2_Vizu.IndexStavu_Cistenie:= 1;
	ELSIF P2_Cistenie.Automat AND P2_Cistenie.STAV.PoINIT THEN
		P2_Vizu.IndexStavu_Cistenie:= 2;
	ELSE
		P2_Vizu.IndexStavu_Cistenie:= 0;
	END_IF

	//Spodný stoper//
	IF P2_SpodnyStoper.Automat AND NOT P2_SpodnyStoper.STAV.PoINIT THEN
		P2_Vizu.IndexStavu_SpodnyStoper:= 1;
	ELSIF P2_SpodnyStoper.Automat AND P2_SpodnyStoper.STAV.PoINIT THEN
		P2_Vizu.IndexStavu_SpodnyStoper:= 2;
	ELSE
		P2_Vizu.IndexStavu_SpodnyStoper:= 0;
	END_IF

END_PROGRAM

PROGRAM _EXIT
	(* Insert code here *)

END_PROGRAM
```

### Program Logical/Program/Pracovisko_2/P2_OvladSafety (IEC)

#### Main.st - Init, cyclic, exit code
```iecst
PROGRAM _INIT
	(* Insert code here *)

END_PROGRAM

PROGRAM _CYCLIC

	//Ovládanie pneuzámku skrutkovačky matice//
	IF Safety.STAV.P2_ZonaMaticovacky_AKTIVNA THEN
		P2_StoperMaticovacky.OUT.Maticovacka_M4_Pneuzamok_ODOMKNI:= TRUE;
	ELSE
		P2_StoperMaticovacky.OUT.Maticovacka_M4_Pneuzamok_ODOMKNI:= FALSE;
	END_IF

	//******************************************Ovládanie zámkov dverí bunky****************************************//
	//Zadné dvere //
	IF P2_Vizu.TL_ZamkniZadneZamky THEN
		IF NOT P2_Pracovisko.STAV.ZadneDvereZamknute AND P2_Pracovisko.IN.ZadneDvereLS_PritomnostAdaptera AND P2_Pracovisko.IN.ZadneDverePS_PritomnostAdaptera THEN
			P2_Pracovisko.OUT.ZadneDvereLS_ZAMKNI:= TRUE;
			P2_Pracovisko.OUT.ZadneDverePS_ZAMKNI:= TRUE;
		ELSIF P2_Pracovisko.STAV.ZadneDvereZamknute THEN
			P2_Pracovisko.OUT.ZadneDvereLS_ZAMKNI:= FALSE;
			P2_Pracovisko.OUT.ZadneDverePS_ZAMKNI:= FALSE;
		END_IF
		P2_Vizu.TL_ZamkniZadneZamky:= FALSE;
	END_IF

	//Predné dvere //
	IF P2_Vizu.TL_ZamkniPredneZamky THEN
		IF NOT P2_Pracovisko.STAV.PredneDvereZamknute AND P2_Pracovisko.IN.PredneDvereLS_PritomnostAdaptera AND P2_Pracovisko.IN.PredneDverePS_PritomnostAdaptera THEN
			P2_Pracovisko.OUT.PredneDvereLS_ZAMKNI:= TRUE;
			P2_Pracovisko.OUT.PredneDverePS_ZAMKNI:= TRUE;
		ELSIF P2_Pracovisko.STAV.PredneDvereZamknute THEN
			P2_Pracovisko.OUT.PredneDvereLS_ZAMKNI:= FALSE;
			P2_Pracovisko.OUT.PredneDverePS_ZAMKNI:= FALSE;
		END_IF
		P2_Vizu.TL_ZamkniPredneZamky:= FALSE;
	END_IF

	//Stav zadné dvere zamknuté//
	IF P2_Pracovisko.OUT.ZadneDvereLS_ZAMKNI AND P2_Pracovisko.OUT.ZadneDverePS_ZAMKNI THEN
		P2_Pracovisko.STAV.ZadneDvereZamknute:= TRUE;
	ELSE
		P2_Pracovisko.STAV.ZadneDvereZamknute:= FALSE;
	END_IF

	//Stav predné dvere zamknuté//
	IF P2_Pracovisko.OUT.PredneDvereLS_ZAMKNI AND P2_Pracovisko.OUT.PredneDverePS_ZAMKNI THEN
		P2_Pracovisko.STAV.PredneDvereZamknute:= TRUE;
	ELSE
		P2_Pracovisko.STAV.PredneDvereZamknute:= FALSE;
	END_IF

	//*****************************************Reset zóny bunky************************************************//
	IF Safety.STAV.Linka_ZonaCS_AKTIVNA AND
		(Safety.STAV.P2_Bunka_Zamky_AKTIVNE OR Safety.STAV.P2_VyblokovanieZamkov_AKTIVNE) AND
		NOT Safety.STAV.P2_ZonaBunky_AKTIVNA AND
		Safety.STAV.P2_Bunka_VstupBariera_AKTIVNA AND
		(Safety.STAV.P3_Bunka_VstupBariera_AKTIVNA OR Safety.STAV.P3_Bunka_Zamky_AKTIVNE)THEN
		Safety.OUT.P2_ResetZonyBunky:= TRUE;
	ELSE
		Safety.OUT.P2_ResetZonyBunky:= FALSE;
	END_IF

END_PROGRAM

PROGRAM _EXIT
	(* Insert code here *)

END_PROGRAM
```

### Program Logical/Program/Pracovisko_2/P2_Mapping_IO (IEC)

#### Main.st - Init, cyclic, exit code
```iecst
PROGRAM _INIT
	(* Insert code here *)

END_PROGRAM

PROGRAM _CYCLIC

	//**********************************************************IO modul Wedmuller**********************************************************************//
	//************Karta AB 2.5 8DI**************//
	P2_Pracovisko.COM_Weidmuller.AB2_5_8DI.0;
	P2_Srobovanie.IN.NapajanieSkrutkovackyM6_OK := P2_Pracovisko.COM_Weidmuller.AB2_5_8DI.1;
	P2_Srobovanie.IN.NapajanieSkrutkovackyM4_OK := P2_Pracovisko.COM_Weidmuller.AB2_5_8DI.2;
	P2_Srobovanie.IN.NapajanieSkrutkovackyM5_OK := P2_Pracovisko.COM_Weidmuller.AB2_5_8DI.3;
	P2_Srobovanie.IN.NapajanieVibrolistyM4_OK := P2_Pracovisko.COM_Weidmuller.AB2_5_8DI.4;
	P2_Srobovanie.IN.NapajanieZasobnikaM6_OK := P2_Pracovisko.COM_Weidmuller.AB2_5_8DI.5;
	P2_Srobovanie.IN.NapajanieZasobnikaM4_OK := P2_Pracovisko.COM_Weidmuller.AB2_5_8DI.6;
	P2_Srobovanie.IN.NapajanieVibrolistyM4_OK := P2_Pracovisko.COM_Weidmuller.AB2_5_8DI.7;

	//************Karta AB 2.6 8DI**************//
	P2_Srobovanie.IN.NapajanieZasobnikaM5_OK := P2_Pracovisko.COM_Weidmuller.AB2_6_8DI.0;
	P2_Zvaranie.IN.NapajanieZvaracky_OK := P2_Pracovisko.COM_Weidmuller.AB2_6_8DI.1;
	P2_Dopravniky.IN.StavRiadeniaDopravBunky_READY := P2_Pracovisko.COM_Weidmuller.AB2_6_8DI.2;
	P2_Dopravniky.IN.StavRiadeniaVratnehoDoprav_READY := P2_Pracovisko.COM_Weidmuller.AB2_6_8DI.3;
	P2_Cistenie.IN.Ionizator_Alarm1 := P2_Pracovisko.COM_Weidmuller.AB2_6_8DI.4;
	P2_Cistenie.IN.Ionizator_Alarm2 := P2_Pracovisko.COM_Weidmuller.AB2_6_8DI.5;
	P2_Cistenie.IN.Ionizator_Alarm3 := P2_Pracovisko.COM_Weidmuller.AB2_6_8DI.6;
	P2_Zvaranie.IN.ZvarackaStav_RUN := P2_Pracovisko.COM_Weidmuller.AB2_6_8DI.7;

	//************Karta AB 2.7 8DI**************//
	P2_Pracovisko.COM_Weidmuller.AB2_7_8DI.0;
	P2_Pracovisko.COM_Weidmuller.AB2_7_8DI.1;
	Safety.IN.Linka_SV_ZonaCS := P2_Pracovisko.COM_Weidmuller.AB2_7_8DI.2;
	Safety.IN.P2_SV_ZonaAutostopRobota := P2_Pracovisko.COM_Weidmuller.AB2_7_8DI.3;
	Safety.IN.P2_SV_ZonaBunky := P2_Pracovisko.COM_Weidmuller.AB2_7_8DI.4;
	Safety.IN.P2_SV_ZonaZakladacaTesnenia := P2_Pracovisko.COM_Weidmuller.AB2_7_8DI.5;
	P2_Pracovisko.COM_Weidmuller.AB2_7_8DI.6;
	Safety.IN.P2_SV_ZonaMaticovacky := P2_Pracovisko.COM_Weidmuller.AB2_7_8DI.7;

	//************Karta AB 2.8 8DI**************//
	P2_Dopravniky.IN.TeplotaMotoraDopravBunky_OK := P2_Pracovisko.COM_Weidmuller.AB2_8_8DI.0;
	P2_Dopravniky.IN.TeplotaMotoraVratnehoDoprav_OK := P2_Pracovisko.COM_Weidmuller.AB2_8_8DI.1;
	P2_Zvaranie.IN.ZvarackaStav_READY := P2_Pracovisko.COM_Weidmuller.AB2_8_8DI.2;
	P2_Pracovisko.COM_Weidmuller.AB2_8_8DI.3;
	P2_Pracovisko.COM_Weidmuller.AB2_8_8DI.4;
	P2_Pracovisko.COM_Weidmuller.AB2_8_8DI.5;
	P2_Pracovisko.COM_Weidmuller.AB2_8_8DI.6;
	P2_Pracovisko.COM_Weidmuller.AB2_8_8DI.7;

	IF P2_Pracovisko.COM_Weidmuller.AB2_8_8DI.6 AND	P2_Pracovisko.COM_Weidmuller.AB2_8_8DI.7 THEN
		Safety.STAV.P2_DvojrucneOvladanie_AKTIVNE:= TRUE;
	ELSE
		Safety.STAV.P2_DvojrucneOvladanie_AKTIVNE:= FALSE;
	END_IF

	//************Karta AB 2.9 8DO***************//
	P2_Pracovisko.COM_Weidmuller.AB2_9_8DO.0 := P2_Pracovisko.OUT.Majak_ZeleneSvetlo_ON;
	P2_Pracovisko.COM_Weidmuller.AB2_9_8DO.1 := P2_Pracovisko.OUT.Majak_OranzoveSvetlo_ON;
	P2_Pracovisko.COM_Weidmuller.AB2_9_8DO.2 := P2_Pracovisko.OUT.Majak_CerveneSvetlo_ON;
	P2_Pracovisko.COM_Weidmuller.AB2_9_8DO.3 := P2_Pracovisko.OUT.Majak_Hukacka_ON;
	P2_Pracovisko.COM_Weidmuller.AB2_9_8DO.4 := P2_StoperMaticovacky.SkrutSet_MaticaM4.OUT.VibropohonZasobnika_RUN;
	P2_Pracovisko.COM_Weidmuller.AB2_9_8DO.5 := P2_Srobovanie.SkrutSet_M6.OUT.VibracnyHrniec.ZapniVibromotor;
	P2_Pracovisko.COM_Weidmuller.AB2_9_8DO.6 := P2_Srobovanie.SkrutSet_M4.OUT.VibropohonZasobnika_RUN;
	P2_Pracovisko.COM_Weidmuller.AB2_9_8DO.7 := P2_Srobovanie.SkrutSet_M4.OUT.VibropohonListy_RUN;

	//************Karta AB 2.10 8DO***************//
	P2_Pracovisko.COM_Weidmuller.AB2_10_8DO.0 := P2_Cistenie.OUT.Ionizator_OFF;
	P2_Pracovisko.COM_Weidmuller.AB2_10_8DO.1 := P2_Zvaranie.OUT.Zvaracka_START;
	P2_Pracovisko.COM_Weidmuller.AB2_10_8DO.2 := P2_Zvaranie.OUT.Zvaracka_RESET;
	P2_Pracovisko.COM_Weidmuller.AB2_10_8DO.3 := P2_Dopravniky.OUT.DopravnikBunky_ON;
	P2_Pracovisko.COM_Weidmuller.AB2_10_8DO.4 := P2_Dopravniky.OUT.VratnyDopravnik_ON;
	P2_Pracovisko.COM_Weidmuller.AB2_10_8DO.5 := P2_ZakladacTesnenia.OUT.LED_DvojrucneOvladanie_ON;
	P2_Pracovisko.COM_Weidmuller.AB2_10_8DO.6:= P2_Pracovisko.OUT.Osvetlenie_CAM10;
	P2_Pracovisko.COM_Weidmuller.AB2_10_8DO.7:= P2_Pracovisko.OUT.Osvetlenie_CAM11;;

	//************Karta AB 2.12 8DO***************//
	P2_Pracovisko.COM_Weidmuller.AB2_12_8DO.0;
	P2_Pracovisko.COM_Weidmuller.AB2_12_8DO.1;
	P2_Pracovisko.COM_Weidmuller.AB2_12_8DO.2:= P2_Pracovisko.OUT.OsvetlenieBunky_ON;;
	P2_Pracovisko.COM_Weidmuller.AB2_12_8DO.3:= P2_Pracovisko.OUT.OsvetleniePracZaklTesnenia_ON;
	P2_Pracovisko.COM_Weidmuller.AB2_12_8DO.4:= P2_Pracovisko.OUT.Osvetlenie_CAM12;
	P2_Pracovisko.COM_Weidmuller.AB2_12_8DO.5:= P2_Pracovisko.OUT.Osvetlenie_CAM1_Svetlo1;
	P2_Pracovisko.COM_Weidmuller.AB2_12_8DO.6:= P2_Pracovisko.OUT.Osvetlenie_CAM1_Svetlo2;
	P2_Pracovisko.COM_Weidmuller.AB2_12_8DO.7:= P2_Srobovanie.SkrutSet_M5.OUT.VibracnyHrniec.ZapniVibromotor;

	//************Karta AB 2.13 8DO***************//
	P2_Pracovisko.COM_Weidmuller.AB2_13_8DO.0:= P2_Pracovisko.OUT.Srobovanie_OsvetleniePaletky_ON;
	P2_Pracovisko.COM_Weidmuller.AB2_13_8DO.1:= P2_Pracovisko.OUT.Srobovanie_BodoveOsvetlenie_ON;
	P2_Pracovisko.COM_Weidmuller.AB2_13_8DO.2;
	P2_Pracovisko.COM_Weidmuller.AB2_13_8DO.3;
	P2_Pracovisko.COM_Weidmuller.AB2_13_8DO.4:= Safety.OUT.Linka_ResetCS;
	P2_Pracovisko.COM_Weidmuller.AB2_13_8DO.5:= Safety.OUT.P2_ResetZonyBunky;
	P2_Pracovisko.COM_Weidmuller.AB2_13_8DO.6;
	P2_Pracovisko.COM_Weidmuller.AB2_13_8DO.7;

	//**************************************************************IO modul Festo**********************************************************************************//

	//**********Modul DM 2.1 4DI4DO**************//
	//Inputs//
	P2_Pracovisko.IN.PredneDvereLS_PritomnostAdaptera := P2_Pracovisko.COM_Festo.DM2_1_4DI[0];
	P2_Pracovisko.IN.PredneDverePS_PritomnostAdaptera := P2_Pracovisko.COM_Festo.DM2_1_4DI[1];
	P2_Pracovisko.IN.ZadneDverePS_PritomnostAdaptera :=  P2_Pracovisko.COM_Festo.DM2_1_4DI[2];
	P2_Pracovisko.IN.ZadneDvereLS_PritomnostAdaptera :=  P2_Pracovisko.COM_Festo.DM2_1_4DI[3];

	//Outputs//
	P2_Pracovisko.COM_Festo.DM2_1_4DO[0]:= P2_Pracovisko.OUT.PredneDvereLS_ZAMKNI;
	P2_Pracovisko.COM_Festo.DM2_1_4DO[1]:=P2_Pracovisko.OUT.PredneDverePS_ZAMKNI;
	P2_Pracovisko.COM_Festo.DM2_1_4DO[2]:= P2_Pracovisko.OUT.ZadneDverePS_ZAMKNI;
	P2_Pracovisko.COM_Festo.DM2_1_4DO[3]:= P2_Pracovisko.OUT.ZadneDvereLS_ZAMKNI;

	//**********Modul DI 2.1 8DI**************//
	P2_Pracovisko.IN.TlakVzduchu_OK := P2_Pracovisko.COM_Festo.DI2_1_8DI[0];
	Safety.IN.P2_SV_PrivodVzduchu_CH1 := P2_Pracovisko.COM_Festo.DI2_1_8DI[1];
	Safety.IN.P2_SV_PrivodVzduchu_CH2 := P2_Pracovisko.COM_Festo.DI2_1_8DI[2];
	P2_ZakladacTesnenia.IN.Pojazd_PritomPowerCP := P2_Pracovisko.COM_Festo.DI2_1_8DI[3];
	P2_ZakladacTesnenia.IN.Kopito_ZakladPoloha := P2_Pracovisko.COM_Festo.DI2_1_8DI[4];
	P2_SpodnyStoper.IN.ZaplnenieDopravnika := P2_Pracovisko.COM_Festo.DI2_1_8DI[5];
	P2_Pracovisko.COM_Festo.DI2_1_8DI[6];
	P2_Pracovisko.COM_Festo.DI2_1_8DI[7];

	//**********Modul DI 2.2 8DI**************//
	P2_Zvaranie.IN.ZvaraniePresunute_VPRAVO := P2_Pracovisko.COM_Festo.DI2_2_8DI[0];
	P2_Zvaranie.IN.ZvaraniePresunute_VLAVO := P2_Pracovisko.COM_Festo.DI2_2_8DI[1];
	P2_Pracovisko.COM_Festo.DI2_2_8DI[2];
	P2_StoperMaticovacky.SkrutSet_MaticaM4.IN.OddelovacOtoceny_VYSTUP := P2_Pracovisko.COM_Festo.DI2_2_8DI[3];
	P2_StoperMaticovacky.SkrutSet_MaticaM4.IN.OddelovacOtoceny_VSTUP := P2_Pracovisko.COM_Festo.DI2_2_8DI[4];
	P2_Srobovanie.SkrutSet_M4.IN.PodavacOtoceny_VSTUP := P2_Pracovisko.COM_Festo.DI2_2_8DI[5];
	P2_Srobovanie.SkrutSet_M4.IN.PodavacOtoceny_VYSTUP := P2_Pracovisko.COM_Festo.DI2_2_8DI[6];
	P2_Pracovisko.COM_Festo.DI2_2_8DI[7];

	//**********Modul DI 2.3 8DI**************//
	P2_Cistenie.IN.Dvere_OTVORENE := P2_Pracovisko.COM_Festo.DI2_3_8DI[0];
	P2_Cistenie.IN.Dvere_ZATVORENE := P2_Pracovisko.COM_Festo.DI2_3_8DI[1];
	P2_Cistenie.IN.Vakum_OK := P2_Pracovisko.COM_Festo.DI2_3_8DI[2];
	P2_Robot.IN.DokStanica_PritomGripraMvCase := P2_Pracovisko.COM_Festo.DI2_3_8DI[3];
	P2_Robot.IN.DokStanica_PritomGripraBusbar45F := P2_Pracovisko.COM_Festo.DI2_3_8DI[4];
	P2_Robot.IN.DokStanica_PritomGripraBusbar5H := P2_Pracovisko.COM_Festo.DI2_3_8DI[5];
	P2_Robot.IN.Model45F_Vakum_OK := P2_Pracovisko.COM_Festo.DI2_3_8DI[6];
	P2_Robot.IN.Model5H_Vakum_OK := P2_Pracovisko.COM_Festo.DI2_3_8DI[7];

	//**********Modul DI 2.4 8DI**************//
	P2_StoperMaticovacky.IN.Centrovanie_ZASUNUTE := P2_Pracovisko.COM_Festo.DI2_4_8DI[0];
	P2_StoperMaticovacky.IN.Centrovanie_VYSUNUTE := P2_Pracovisko.COM_Festo.DI2_4_8DI[1];
	P2_StoperSrobovania.IN.Centrovanie_VYSUNUTE := P2_Pracovisko.COM_Festo.DI2_4_8DI[2];
	P2_AkumulacnyStoper.IN.PritomnostPaletky := P2_Pracovisko.COM_Festo.DI2_4_8DI[3];
	P2_StoperZvarania.IN.Centrovanie_VYSUNUTE := P2_Pracovisko.COM_Festo.DI2_4_8DI[4];
	P2_StoperSrobovania.IN.Centrovanie_ZASUNUTE := P2_Pracovisko.COM_Festo.DI2_4_8DI[5];
	P2_SpodnyStoper.IN.PritomnostPaletky := P2_Pracovisko.COM_Festo.DI2_4_8DI[6];
	P2_StoperZvarania.IN.Centrovanie_ZASUNUTE := P2_Pracovisko.COM_Festo.DI2_4_8DI[7];

	//**********Modul DI 2.5 8DI**************//
	P2_Srobovanie.SkrutSet_M5.IN.VibracnyHrniec.PritomnostSkrutiekVHrnci := P2_Pracovisko.COM_Festo.DI2_5_8DI[0];
	P2_Srobovanie.SkrutSet_M5.IN.VibracnyHrniec.VibracnaListaZaplnena := P2_Pracovisko.COM_Festo.DI2_5_8DI[1];
	P2_Srobovanie.SkrutSet_M5.IN.Brzda.PreletSkrutky := P2_Pracovisko.COM_Festo.DI2_5_8DI[2];
	P2_Srobovanie.SkrutSet_M5.IN.Brzda.PodajSkrutku := P2_Pracovisko.COM_Festo.DI2_5_8DI[3];
	P2_Srobovanie.SkrutSet_M5.IN.Brzda.ZakladnaPoloha := P2_Pracovisko.COM_Festo.DI2_5_8DI[4];
	P2_Srobovanie.SkrutSet_M5.IN.Brzda.SkrutkaPritomnaVBrzde := P2_Pracovisko.COM_Festo.DI2_5_8DI[5];
	P2_Srobovanie.SkrutSet_M5.IN.VibracnyHrniec.PreletovySnimac := P2_Pracovisko.COM_Festo.DI2_5_8DI[6];
	P2_Srobovanie.IN.Skrutkovacka_M5_ZASUNUTA := P2_Pracovisko.COM_Festo.DI2_5_8DI[7];

	//**********Modul DI 2.6 8DI**************//
	P2_StoperMaticovacky.SkrutSet_MaticaM4.IN.ZasobnikMaticPrazdny := P2_Pracovisko.COM_Festo.DI2_6_8DI[0];
	P2_StoperMaticovacky.SkrutSet_MaticaM4.IN.ZaplnenieListyZasobnika := P2_Pracovisko.COM_Festo.DI2_6_8DI[1];
	P2_StoperMaticovacky.SkrutSet_MaticaM4.IN.Oddelovac_SnimPrechoduMatice := P2_Pracovisko.COM_Festo.DI2_6_8DI[2];
	P2_StoperMaticovacky.SkrutSet_MaticaM4.IN.PritomnostMaticeNaVystupe :=  P2_Pracovisko.COM_Festo.DI2_6_8DI[3];
	P2_StoperMaticovacky.SkrutSet_MaticaM4.IN.PodavacMatice_ZASUNUTY :=  P2_Pracovisko.COM_Festo.DI2_6_8DI[4];
	P2_StoperMaticovacky.SkrutSet_MaticaM4.IN.PodavacMatice_VYSUNUTY := P2_Pracovisko.COM_Festo.DI2_6_8DI[5];
	P2_StoperMaticovacky.SkrutSet_MaticaM4.IN.Podavac_SnimPrechoduMatice := P2_Pracovisko.COM_Festo.DI2_6_8DI[6];
	P2_StoperMaticovacky.IN.Maticovacka_M4_ZASUNUTA := P2_Pracovisko.COM_Festo.DI2_6_8DI[7];

	//**********Modul DI 2.7 8DI**************//
	P2_Srobovanie.SkrutSet_M4.IN.ZasobnikSkrutiekPrazdny := P2_Pracovisko.COM_Festo.DI2_7_8DI[0];
	P2_Srobovanie.SkrutSet_M4.IN.ZaplnenieListyZasobnika := P2_Pracovisko.COM_Festo.DI2_7_8DI[1];
	P2_Srobovanie.SkrutSet_M4.IN.ZaplnenieVibrolisty_MAX := P2_Pracovisko.COM_Festo.DI2_7_8DI[2];
	P2_Srobovanie.SkrutSet_M4.IN.ZaplnenieVibrolisty_MIN := P2_Pracovisko.COM_Festo.DI2_7_8DI[3];
	P2_Srobovanie.SkrutSet_M4.IN.Podavac_SkrutkaNaVstupe := P2_Pracovisko.COM_Festo.DI2_7_8DI[4];
	P2_Srobovanie.SkrutSet_M4.IN.Podavac_SkrutkaNaVystupe := P2_Pracovisko.COM_Festo.DI2_7_8DI[5];
	P2_Srobovanie.IN.Skrutkovacka_M4_Vakum_OK := P2_Pracovisko.COM_Festo.DI2_7_8DI[6];
	P2_Pracovisko.COM_Festo.DI2_7_8DI[7];

	//**********Modul DI 2.8 8DI**************//
	P2_Srobovanie.SkrutSet_M6.IN.VibracnyHrniec.PritomnostSkrutiekVHrnci := P2_Pracovisko.COM_Festo.DI2_8_8DI[0];
	P2_Srobovanie.SkrutSet_M6.IN.VibracnyHrniec.VibracnaListaZaplnena := P2_Pracovisko.COM_Festo.DI2_8_8DI[1];
	P2_Srobovanie.SkrutSet_M6.IN.Brzda.PreletSkrutky := P2_Pracovisko.COM_Festo.DI2_8_8DI[2];
	P2_Srobovanie.SkrutSet_M6.IN.Brzda.PodajSkrutku := P2_Pracovisko.COM_Festo.DI2_8_8DI[3];
	P2_Srobovanie.SkrutSet_M6.IN.Brzda.ZakladnaPoloha := P2_Pracovisko.COM_Festo.DI2_8_8DI[4];
	P2_Srobovanie.SkrutSet_M6.IN.Brzda.SkrutkaPritomnaVBrzde := P2_Pracovisko.COM_Festo.DI2_8_8DI[5];
	P2_Srobovanie.SkrutSet_M6.IN.VibracnyHrniec.PreletovySnimac := P2_Pracovisko.COM_Festo.DI2_8_8DI[6];
	P2_Srobovanie.IN.Skrutkovacka_M6_ZASUNUTA := P2_Pracovisko.COM_Festo.DI2_8_8DI[7];

	//********Modul DS 2.1 IO link Port 0 - IO_Modul Balluff***************//
	//Inputs//
	P2_Pracovisko.COM_Festo.DS2_1_Port0_IN[0].0;  //IS2.36
	P2_Pracovisko.COM_Festo.DS2_1_Port0_IN[0].1;  //IS2.37
	P2_Pracovisko.COM_Festo.DS2_1_Port0_IN[0].2;  //IS2.38
	P2_Pracovisko.COM_Festo.DS2_1_Port0_IN[0].3;
	P2_Pracovisko.COM_Festo.DS2_1_Port0_IN[0].4;
	P2_Pracovisko.COM_Festo.DS2_1_Port0_IN[0].5;
	P2_Robot.IN.KodGripra_Bit0:= P2_Pracovisko.COM_Festo.DS2_1_Port0_IN[0].6;
	P2_Robot.IN.KodGripra_Bit1:= P2_Pracovisko.COM_Festo.DS2_1_Port0_IN[0].7;

	P2_Pracovisko.COM_Festo.DS2_1_Port0_IN[1].0;
	P2_Pracovisko.COM_Festo.DS2_1_Port0_IN[1].1;
	P2_Pracovisko.COM_Festo.DS2_1_Port0_IN[1].2;
	P2_Pracovisko.COM_Festo.DS2_1_Port0_IN[1].3;
	P2_Pracovisko.COM_Festo.DS2_1_Port0_IN[1].4;
	P2_Pracovisko.COM_Festo.DS2_1_Port0_IN[1].5;
	P2_Pracovisko.COM_Festo.DS2_1_Port0_IN[1].6;
	P2_Pracovisko.COM_Festo.DS2_1_Port0_IN[1].7;

	//Outputs//
	P2_Pracovisko.COM_Festo.DS2_1_Port0_OUT[0].0;
	P2_Pracovisko.COM_Festo.DS2_1_Port0_OUT[0].1;
	P2_Pracovisko.COM_Festo.DS2_1_Port0_OUT[0].2;
	P2_Pracovisko.COM_Festo.DS2_1_Port0_OUT[0].3;
	P2_Pracovisko.COM_Festo.DS2_1_Port0_OUT[0].4;
	P2_Pracovisko.COM_Festo.DS2_1_Port0_OUT[0].5;
	P2_Pracovisko.COM_Festo.DS2_1_Port0_OUT[0].6;
	P2_Pracovisko.COM_Festo.DS2_1_Port0_OUT[0].7;

	P2_Pracovisko.COM_Festo.DS2_1_Port0_OUT[1].0;
	P2_Pracovisko.COM_Festo.DS2_1_Port0_OUT[1].1;
	P2_Pracovisko.COM_Festo.DS2_1_Port0_OUT[1].2;
	P2_Pracovisko.COM_Festo.DS2_1_Port0_OUT[1].3;
	P2_Pracovisko.COM_Festo.DS2_1_Port0_OUT[1].4;
	P2_Pracovisko.COM_Festo.DS2_1_Port0_OUT[1].5;
	P2_Pracovisko.COM_Festo.DS2_1_Port0_OUT[1].6;
	P2_Pracovisko.COM_Festo.DS2_1_Port0_OUT[1].7;

	//*************Modul DS 2.1 IO link Port 1 - Snímač vysunutia skrutkovačky M5*********************//
	//Inputs//
	Convert_0.IN_Byte1:= P2_Pracovisko.COM_Festo.DS2_1_Port1_IN[0];
	Convert_0.IN_Byte0:= P2_Pracovisko.COM_Festo.DS2_1_Port1_IN[1];

	P2_Srobovanie.PAR.Skrutkov_M5_AktualHodnVysunutia:= Convert_0.OUT_UINT;
	Convert_0();

	//*************Modul DS 2.1 IO link Port 2 - Snímač vysunutia skrutkovačky M6*********************//
	//Inputs//
	Convert_1.IN_Byte1:= P2_Pracovisko.COM_Festo.DS2_1_Port2_IN[0];
	Convert_1.IN_Byte0:= P2_Pracovisko.COM_Festo.DS2_1_Port2_IN[1];

	P2_Srobovanie.PAR.Skrutkov_M6_AktualHodnVysunutia:= Convert_1.OUT_UINT;
	Convert_1();

	//*************Modul DS 2.1 IO link Port 3 - Snímač otvorenia zatvorenia gripra robota*********************//
	//Inputs//
	Convert_2.IN_Byte0:= P2_Pracovisko.COM_Festo.DS2_1_Port3_IN[0];
	Convert_2.IN_Byte1:= P2_Pracovisko.COM_Festo.DS2_1_Port3_IN[1];

	IF P2_Robot.IN.KodGripra_Bit0 AND P2_Robot.IN.KodGripra_Bit1 THEN
		P2_Robot.PAR.Griper_Busbary45F_HodnOtvorenia:= 0;
		P2_Robot.PAR.Griper_Busbary5H_HodnOtvorenia:= Convert_2.OUT_UINT;
	ELSIF NOT P2_Robot.IN.KodGripra_Bit0 AND P2_Robot.IN.KodGripra_Bit1 THEN
		P2_Robot.PAR.Griper_Busbary5H_HodnOtvorenia:= 0;
		P2_Robot.PAR.Griper_Busbary45F_HodnOtvorenia:= Convert_2.OUT_UINT;
	ELSE
		P2_Robot.PAR.Griper_Busbary5H_HodnOtvorenia:= 0;
		P2_Robot.PAR.Griper_Busbary45F_HodnOtvorenia:= 0;
	END_IF

	Convert_2();

	//Typ gripra//
	P2_Robot.IN.TypGripra_45F:= NOT P2_Robot.IN.KodGripra_Bit0 AND P2_Robot.IN.KodGripra_Bit1;
	P2_Robot.IN.TypGripra_5H:= P2_Robot.IN.KodGripra_Bit0 AND P2_Robot.IN.KodGripra_Bit1;
	P2_Robot.IN.TypGripra_MvCase:= P2_Robot.IN.KodGripra_Bit0 AND NOT P2_Robot.IN.KodGripra_Bit1;

	//Stavy gripra 45F//
	IF P2_Robot.IN.TypGripra_45F THEN
		IF P2_Robot.PAR.Griper_Busbary45F_HodnOtvorenia < 17500 THEN
			P2_Robot.IN.Griper45F_Zatvoreny:= FALSE;
			P2_Robot.IN.Griper45F_DrziBusbary:= FALSE;
			P2_Robot.IN.Griper45F_Otvoreny:= TRUE;
		ELSIF P2_Robot.PAR.Griper_Busbary45F_HodnOtvorenia > 44000 THEN
			P2_Robot.IN.Griper45F_Otvoreny:= FALSE;
			P2_Robot.IN.Griper45F_DrziBusbary:= FALSE;
			P2_Robot.IN.Griper45F_Zatvoreny:= TRUE;
		ELSIF P2_Robot.PAR.Griper_Busbary45F_HodnOtvorenia > 21000 AND P2_Robot.PAR.Griper_Busbary45F_HodnOtvorenia < 31000 THEN
			P2_Robot.IN.Griper45F_Otvoreny:= FALSE;
			P2_Robot.IN.Griper45F_Zatvoreny:= FALSE;
			P2_Robot.IN.Griper45F_DrziBusbary:= TRUE;
		ELSE
			P2_Robot.IN.Griper45F_Otvoreny:= FALSE;
			P2_Robot.IN.Griper45F_Zatvoreny:= FALSE;
			P2_Robot.IN.Griper45F_DrziBusbary:= FALSE;
		END_IF
	ELSE
		P2_Robot.IN.Griper45F_Otvoreny:= FALSE;
		P2_Robot.IN.Griper45F_Zatvoreny:= FALSE;
		P2_Robot.IN.Griper45F_DrziBusbary:= FALSE;
	END_IF

	//Stavy gripra 5H//
	IF P2_Robot.IN.TypGripra_5H THEN
		IF P2_Robot.PAR.Griper_Busbary5H_HodnOtvorenia < 19600 THEN
			P2_Robot.IN.Griper5H_Zatvoreny:= FALSE;
			P2_Robot.IN.Griper5H_DrziBusbary:= FALSE;
			P2_Robot.IN.Griper5H_Otvoreny:= TRUE;
		ELSIF P2_Robot.PAR.Griper_Busbary5H_HodnOtvorenia > 50000 THEN
			P2_Robot.IN.Griper5H_Otvoreny:= FALSE;
			P2_Robot.IN.Griper5H_DrziBusbary:= FALSE;
			P2_Robot.IN.Griper5H_Zatvoreny:= TRUE;
		ELSIF P2_Robot.PAR.Griper_Busbary5H_HodnOtvorenia > 21000 AND P2_Robot.PAR.Griper_Busbary5H_HodnOtvorenia < 34000 THEN
			P2_Robot.IN.Griper5H_Otvoreny:= FALSE;
			P2_Robot.IN.Griper5H_Zatvoreny:= FALSE;
			P2_Robot.IN.Griper5H_DrziBusbary:= TRUE;
		ELSE
			P2_Robot.IN.Griper5H_Otvoreny:= FALSE;
			P2_Robot.IN.Griper5H_Zatvoreny:= FALSE;
			P2_Robot.IN.Griper5H_DrziBusbary:= FALSE;
		END_IF
	ELSE
		P2_Robot.IN.Griper5H_Otvoreny:= FALSE;
		P2_Robot.IN.Griper5H_Zatvoreny:= FALSE;
		P2_Robot.IN.Griper5H_DrziBusbary:= FALSE;
	END_IF

	//Stavy gripra MV case//
	IF P2_Robot.IN.TypGripra_MvCase THEN
		IF NOT P2_Pracovisko.COM_Festo.DS2_1_Port0_IN[0].0 AND P2_Pracovisko.COM_Festo.DS2_1_Port0_IN[0].1 AND NOT P2_Pracovisko.COM_Festo.DS2_1_Port0_IN[0].2 THEN
			P2_Robot.IN.GriperMvCase_DrziPowerCP:= FALSE;
			P2_Robot.IN.GriperMvCase_DrziMvCase:= FALSE;
			P2_Robot.IN.GriperMvCase_Zatvoreny:= FALSE;
			P2_Robot.IN.GriperMvCase_Otvoreny:= TRUE;
		ELSIF P2_Pracovisko.COM_Festo.DS2_1_Port0_IN[0].0 AND NOT P2_Pracovisko.COM_Festo.DS2_1_Port0_IN[0].1 AND NOT P2_Pracovisko.COM_Festo.DS2_1_Port0_IN[0].2 THEN
			P2_Robot.IN.GriperMvCase_DrziPowerCP:= FALSE;
			P2_Robot.IN.GriperMvCase_DrziMvCase:= FALSE;
			P2_Robot.IN.GriperMvCase_Zatvoreny:= TRUE;
			P2_Robot.IN.GriperMvCase_Otvoreny:= FALSE;
		ELSIF P2_Pracovisko.COM_Festo.DS2_1_Port0_IN[0].0 AND NOT P2_Pracovisko.COM_Festo.DS2_1_Port0_IN[0].1 AND P2_Pracovisko.COM_Festo.DS2_1_Port0_IN[0].2 THEN
			P2_Robot.IN.GriperMvCase_DrziPowerCP:= FALSE;
			P2_Robot.IN.GriperMvCase_DrziMvCase:= TRUE;
			P2_Robot.IN.GriperMvCase_Zatvoreny:= FALSE;
			P2_Robot.IN.GriperMvCase_Otvoreny:= FALSE;
		ELSIF P2_Pracovisko.COM_Festo.DS2_1_Port0_IN[0].0 AND P2_Pracovisko.COM_Festo.DS2_1_Port0_IN[0].1 AND NOT P2_Pracovisko.COM_Festo.DS2_1_Port0_IN[0].2 THEN
			P2_Robot.IN.GriperMvCase_DrziPowerCP:= TRUE;
			P2_Robot.IN.GriperMvCase_DrziMvCase:= FALSE;
			P2_Robot.IN.GriperMvCase_Zatvoreny:= FALSE;
			P2_Robot.IN.GriperMvCase_Otvoreny:= FALSE;
		ELSE
			P2_Robot.IN.GriperMvCase_DrziPowerCP:= FALSE;
			P2_Robot.IN.GriperMvCase_DrziMvCase:= FALSE;
			P2_Robot.IN.GriperMvCase_Zatvoreny:= FALSE;
			P2_Robot.IN.GriperMvCase_Otvoreny:= FALSE;
		END_IF
	ELSE
		P2_Robot.IN.GriperMvCase_DrziPowerCP:= FALSE;
		P2_Robot.IN.GriperMvCase_DrziMvCase:= FALSE;
		P2_Robot.IN.GriperMvCase_Zatvoreny:= FALSE;
		P2_Robot.IN.GriperMvCase_Otvoreny:= FALSE;
	END_IF

	//********Modul DS 2.2 IO link Port 0 - RFID snímač paletky zakladač tesnenia**************//
	//Inputs//
	P2_StoperZaklTesnenia.RFID_hlava.Mapping_IN[0]:= P2_Pracovisko.COM_Festo.DS2_2_Port0_IN[0];
	P2_StoperZaklTesnenia.RFID_hlava.Mapping_IN[1]:= P2_Pracovisko.COM_Festo.DS2_2_Port0_IN[1];
	P2_StoperZaklTesnenia.RFID_hlava.Mapping_IN[2]:= P2_Pracovisko.COM_Festo.DS2_2_Port0_IN[2];
	P2_StoperZaklTesnenia.RFID_hlava.Mapping_IN[3]:= P2_Pracovisko.COM_Festo.DS2_2_Port0_IN[3];
	P2_StoperZaklTesnenia.RFID_hlava.Mapping_IN[4]:= P2_Pracovisko.COM_Festo.DS2_2_Port0_IN[4];
	P2_StoperZaklTesnenia.RFID_hlava.Mapping_IN[5]:= P2_Pracovisko.COM_Festo.DS2_2_Port0_IN[5];
	P2_StoperZaklTesnenia.RFID_hlava.Mapping_IN[6]:= P2_Pracovisko.COM_Festo.DS2_2_Port0_IN[6];
	P2_StoperZaklTesnenia.RFID_hlava.Mapping_IN[7]:= P2_Pracovisko.COM_Festo.DS2_2_Port0_IN[7];

	//Outputs//
	P2_Pracovisko.COM_Festo.DS2_2_Port0_OUT[0]:= P2_StoperZaklTesnenia.RFID_hlava.Mapping_OUT[0];
	P2_Pracovisko.COM_Festo.DS2_2_Port0_OUT[1]:= P2_StoperZaklTesnenia.RFID_hlava.Mapping_OUT[1];
	P2_Pracovisko.COM_Festo.DS2_2_Port0_OUT[2]:= P2_StoperZaklTesnenia.RFID_hlava.Mapping_OUT[2];
	P2_Pracovisko.COM_Festo.DS2_2_Port0_OUT[3]:= P2_StoperZaklTesnenia.RFID_hlava.Mapping_OUT[3];
	P2_Pracovisko.COM_Festo.DS2_2_Port0_OUT[4]:= P2_StoperZaklTesnenia.RFID_hlava.Mapping_OUT[4];
	P2_Pracovisko.COM_Festo.DS2_2_Port0_OUT[5]:= P2_StoperZaklTesnenia.RFID_hlava.Mapping_OUT[5];
	P2_Pracovisko.COM_Festo.DS2_2_Port0_OUT[6]:= P2_StoperZaklTesnenia.RFID_hlava.Mapping_OUT[6];
	P2_Pracovisko.COM_Festo.DS2_2_Port0_OUT[7]:= P2_StoperZaklTesnenia.RFID_hlava.Mapping_OUT[7];

	//********Modul DS 2.2 IO link Port 1 - RFID snímač paletky maticovačka**************//
	//Inputs//
	P2_StoperMaticovacky.RFID_hlava.Mapping_IN[0]:= P2_Pracovisko.COM_Festo.DS2_2_Port1_IN[0];
	P2_StoperMaticovacky.RFID_hlava.Mapping_IN[1]:= P2_Pracovisko.COM_Festo.DS2_2_Port1_IN[1];
	P2_StoperMaticovacky.RFID_hlava.Mapping_IN[2]:= P2_Pracovisko.COM_Festo.DS2_2_Port1_IN[2];
	P2_StoperMaticovacky.RFID_hlava.Mapping_IN[3]:= P2_Pracovisko.COM_Festo.DS2_2_Port1_IN[3];
	P2_StoperMaticovacky.RFID_hlava.Mapping_IN[4]:= P2_Pracovisko.COM_Festo.DS2_2_Port1_IN[4];
	P2_StoperMaticovacky.RFID_hlava.Mapping_IN[5]:= P2_Pracovisko.COM_Festo.DS2_2_Port1_IN[5];
	P2_StoperMaticovacky.RFID_hlava.Mapping_IN[6]:= P2_Pracovisko.COM_Festo.DS2_2_Port1_IN[6];
	P2_StoperMaticovacky.RFID_hlava.Mapping_IN[7]:= P2_Pracovisko.COM_Festo.DS2_2_Port1_IN[7];

	//Outputs//
	P2_Pracovisko.COM_Festo.DS2_2_Port1_OUT[0]:= P2_StoperMaticovacky.RFID_hlava.Mapping_OUT[0];
	P2_Pracovisko.COM_Festo.DS2_2_Port1_OUT[1]:= P2_StoperMaticovacky.RFID_hlava.Mapping_OUT[1];
	P2_Pracovisko.COM_Festo.DS2_2_Port1_OUT[2]:= P2_StoperMaticovacky.RFID_hlava.Mapping_OUT[2];
	P2_Pracovisko.COM_Festo.DS2_2_Port1_OUT[3]:= P2_StoperMaticovacky.RFID_hlava.Mapping_OUT[3];
	P2_Pracovisko.COM_Festo.DS2_2_Port1_OUT[4]:= P2_StoperMaticovacky.RFID_hlava.Mapping_OUT[4];
	P2_Pracovisko.COM_Festo.DS2_2_Port1_OUT[5]:= P2_StoperMaticovacky.RFID_hlava.Mapping_OUT[5];
	P2_Pracovisko.COM_Festo.DS2_2_Port1_OUT[6]:= P2_StoperMaticovacky.RFID_hlava.Mapping_OUT[6];
	P2_Pracovisko.COM_Festo.DS2_2_Port1_OUT[7]:= P2_StoperMaticovacky.RFID_hlava.Mapping_OUT[7];

	//********Modul DS 2.2 IO link Port 2 - RFID snímač paletky šrobovanie**************//
	//Inputs//
	P2_StoperSrobovania.RFID_hlava.Mapping_IN[0]:= P2_Pracovisko.COM_Festo.DS2_2_Port2_IN[0];
	P2_StoperSrobovania.RFID_hlava.Mapping_IN[1]:= P2_Pracovisko.COM_Festo.DS2_2_Port2_IN[1];
	P2_StoperSrobovania.RFID_hlava.Mapping_IN[2]:= P2_Pracovisko.COM_Festo.DS2_2_Port2_IN[2];
	P2_StoperSrobovania.RFID_hlava.Mapping_IN[3]:= P2_Pracovisko.COM_Festo.DS2_2_Port2_IN[3];
	P2_StoperSrobovania.RFID_hlava.Mapping_IN[4]:= P2_Pracovisko.COM_Festo.DS2_2_Port2_IN[4];
	P2_StoperSrobovania.RFID_hlava.Mapping_IN[5]:= P2_Pracovisko.COM_Festo.DS2_2_Port2_IN[5];
	P2_StoperSrobovania.RFID_hlava.Mapping_IN[6]:= P2_Pracovisko.COM_Festo.DS2_2_Port2_IN[6];
	P2_StoperSrobovania.RFID_hlava.Mapping_IN[7]:= P2_Pracovisko.COM_Festo.DS2_2_Port2_IN[7];

	//Outputs//
	P2_Pracovisko.COM_Festo.DS2_2_Port2_OUT[0]:= P2_StoperSrobovania.RFID_hlava.Mapping_OUT[0];
	P2_Pracovisko.COM_Festo.DS2_2_Port2_OUT[1]:= P2_StoperSrobovania.RFID_hlava.Mapping_OUT[1];
	P2_Pracovisko.COM_Festo.DS2_2_Port2_OUT[2]:= P2_StoperSrobovania.RFID_hlava.Mapping_OUT[2];
	P2_Pracovisko.COM_Festo.DS2_2_Port2_OUT[3]:= P2_StoperSrobovania.RFID_hlava.Mapping_OUT[3];
	P2_Pracovisko.COM_Festo.DS2_2_Port2_OUT[4]:= P2_StoperSrobovania.RFID_hlava.Mapping_OUT[4];
	P2_Pracovisko.COM_Festo.DS2_2_Port2_OUT[5]:= P2_StoperSrobovania.RFID_hlava.Mapping_OUT[5];
	P2_Pracovisko.COM_Festo.DS2_2_Port2_OUT[6]:= P2_StoperSrobovania.RFID_hlava.Mapping_OUT[6];
	P2_Pracovisko.COM_Festo.DS2_2_Port2_OUT[7]:= P2_StoperSrobovania.RFID_hlava.Mapping_OUT[7];

	//********Modul DS 2.2 IO link Port 3 - RFID snímač paletky zváranie**************//
	//Inputs//
	P2_StoperZvarania.RFID_hlava.Mapping_IN[0]:= P2_Pracovisko.COM_Festo.DS2_2_Port3_IN[0];
	P2_StoperZvarania.RFID_hlava.Mapping_IN[1]:= P2_Pracovisko.COM_Festo.DS2_2_Port3_IN[1];
	P2_StoperZvarania.RFID_hlava.Mapping_IN[2]:= P2_Pracovisko.COM_Festo.DS2_2_Port3_IN[2];
	P2_StoperZvarania.RFID_hlava.Mapping_IN[3]:= P2_Pracovisko.COM_Festo.DS2_2_Port3_IN[3];
	P2_StoperZvarania.RFID_hlava.Mapping_IN[4]:= P2_Pracovisko.COM_Festo.DS2_2_Port3_IN[4];
	P2_StoperZvarania.RFID_hlava.Mapping_IN[5]:= P2_Pracovisko.COM_Festo.DS2_2_Port3_IN[5];
	P2_StoperZvarania.RFID_hlava.Mapping_IN[6]:= P2_Pracovisko.COM_Festo.DS2_2_Port3_IN[6];
	P2_StoperZvarania.RFID_hlava.Mapping_IN[7]:= P2_Pracovisko.COM_Festo.DS2_2_Port3_IN[7];

	//Outputs//
	P2_Pracovisko.COM_Festo.DS2_2_Port3_OUT[0]:= P2_StoperZvarania.RFID_hlava.Mapping_OUT[0];
	P2_Pracovisko.COM_Festo.DS2_2_Port3_OUT[1]:= P2_StoperZvarania.RFID_hlava.Mapping_OUT[1];
	P2_Pracovisko.COM_Festo.DS2_2_Port3_OUT[2]:= P2_StoperZvarania.RFID_hlava.Mapping_OUT[2];
	P2_Pracovisko.COM_Festo.DS2_2_Port3_OUT[3]:= P2_StoperZvarania.RFID_hlava.Mapping_OUT[3];
	P2_Pracovisko.COM_Festo.DS2_2_Port3_OUT[4]:= P2_StoperZvarania.RFID_hlava.Mapping_OUT[4];
	P2_Pracovisko.COM_Festo.DS2_2_Port3_OUT[5]:= P2_StoperZvarania.RFID_hlava.Mapping_OUT[5];
	P2_Pracovisko.COM_Festo.DS2_2_Port3_OUT[6]:= P2_StoperZvarania.RFID_hlava.Mapping_OUT[6];
	P2_Pracovisko.COM_Festo.DS2_2_Port3_OUT[7]:= P2_StoperZvarania.RFID_hlava.Mapping_OUT[7];

	//*************Modul DS 2.3 IO link Port 0 - Banner*********************//
	//Inputs//
	P2_StoperZaklTesnenia.Banner.Mapping_IN[0]:= P2_Pracovisko.COM_Festo.DS2_3_Port0_IN[0];
	P2_StoperZaklTesnenia.Banner.Mapping_IN[1]:= P2_Pracovisko.COM_Festo.DS2_3_Port0_IN[1];
	P2_StoperZaklTesnenia.Banner.Mapping_IN[2]:= P2_Pracovisko.COM_Festo.DS2_3_Port0_IN[2];
	P2_StoperZaklTesnenia.Banner.Mapping_IN[3]:= P2_Pracovisko.COM_Festo.DS2_3_Port0_IN[3];
	P2_StoperZaklTesnenia.Banner.Mapping_IN[4]:= P2_Pracovisko.COM_Festo.DS2_3_Port0_IN[4];
	P2_StoperZaklTesnenia.Banner.Mapping_IN[5]:= P2_Pracovisko.COM_Festo.DS2_3_Port0_IN[5];
	P2_StoperZaklTesnenia.Banner.Mapping_IN[6]:= P2_Pracovisko.COM_Festo.DS2_3_Port0_IN[6];
	P2_StoperZaklTesnenia.Banner.Mapping_IN[7]:= P2_Pracovisko.COM_Festo.DS2_3_Port0_IN[7];
	P2_StoperZaklTesnenia.Banner.Mapping_IN[8]:= P2_Pracovisko.COM_Festo.DS2_3_Port0_IN[8];
	P2_StoperZaklTesnenia.Banner.Mapping_IN[9]:= P2_Pracovisko.COM_Festo.DS2_3_Port0_IN[9];
	P2_StoperZaklTesnenia.Banner.Mapping_IN[10]:= P2_Pracovisko.COM_Festo.DS2_3_Port0_IN[10];
	P2_StoperZaklTesnenia.Banner.Mapping_IN[11]:= P2_Pracovisko.COM_Festo.DS2_3_Port0_IN[11];
	P2_StoperZaklTesnenia.Banner.Mapping_IN[12]:= P2_Pracovisko.COM_Festo.DS2_3_Port0_IN[12];
	P2_StoperZaklTesnenia.Banner.Mapping_IN[13]:= P2_Pracovisko.COM_Festo.DS2_3_Port0_IN[13];
	P2_StoperZaklTesnenia.Banner.Mapping_IN[14]:= P2_Pracovisko.COM_Festo.DS2_3_Port0_IN[14];
	P2_StoperZaklTesnenia.Banner.Mapping_IN[15]:= P2_Pracovisko.COM_Festo.DS2_3_Port0_IN[15];

	//Outputs//
	P2_Pracovisko.COM_Festo.DS2_3_Port0_OUT[0]:= P2_StoperZaklTesnenia.Banner.Mapping_OUT[0];
	P2_Pracovisko.COM_Festo.DS2_3_Port0_OUT[1]:= P2_StoperZaklTesnenia.Banner.Mapping_OUT[1];
	P2_Pracovisko.COM_Festo.DS2_3_Port0_OUT[2]:= P2_StoperZaklTesnenia.Banner.Mapping_OUT[2];
	P2_Pracovisko.COM_Festo.DS2_3_Port0_OUT[3]:= P2_StoperZaklTesnenia.Banner.Mapping_OUT[3];
	P2_Pracovisko.COM_Festo.DS2_3_Port0_OUT[4]:= P2_StoperZaklTesnenia.Banner.Mapping_OUT[4];
	P2_Pracovisko.COM_Festo.DS2_3_Port0_OUT[5]:= P2_StoperZaklTesnenia.Banner.Mapping_OUT[5];
	P2_Pracovisko.COM_Festo.DS2_3_Port0_OUT[6]:= P2_StoperZaklTesnenia.Banner.Mapping_OUT[6];
	P2_Pracovisko.COM_Festo.DS2_3_Port0_OUT[7]:= P2_StoperZaklTesnenia.Banner.Mapping_OUT[7];
	P2_Pracovisko.COM_Festo.DS2_3_Port0_OUT[8]:= P2_StoperZaklTesnenia.Banner.Mapping_OUT[8];
	P2_Pracovisko.COM_Festo.DS2_3_Port0_OUT[9]:= P2_StoperZaklTesnenia.Banner.Mapping_OUT[9];
	P2_Pracovisko.COM_Festo.DS2_3_Port0_OUT[10]:= P2_StoperZaklTesnenia.Banner.Mapping_OUT[10];
	P2_Pracovisko.COM_Festo.DS2_3_Port0_OUT[11]:= P2_StoperZaklTesnenia.Banner.Mapping_OUT[11];
	P2_Pracovisko.COM_Festo.DS2_3_Port0_OUT[12]:= P2_StoperZaklTesnenia.Banner.Mapping_OUT[12];
	P2_Pracovisko.COM_Festo.DS2_3_Port0_OUT[13]:= P2_StoperZaklTesnenia.Banner.Mapping_OUT[13];
	P2_Pracovisko.COM_Festo.DS2_3_Port0_OUT[14]:= P2_StoperZaklTesnenia.Banner.Mapping_OUT[14];
	P2_Pracovisko.COM_Festo.DS2_3_Port0_OUT[15]:= P2_StoperZaklTesnenia.Banner.Mapping_OUT[15];

	//*************Modul DS 2.3 IO link Port 1 - Snímač vysunutia maticovačky M4*********************//
	//Inputs//
	Convert_3.IN_Byte1:= P2_Pracovisko.COM_Festo.DS2_3_Port1_IN[0];
	Convert_3.IN_Byte0:= P2_Pracovisko.COM_Festo.DS2_3_Port1_IN[1];

	P2_StoperMaticovacky.PAR.Maticov_M4_AktualHodnVysunutia:= Convert_3.OUT_UINT;
	Convert_3();

	//************************************Ventilový terminál*******************************************//

	//0-7
	P2_Pracovisko.COM_VentilovyTerminal[0].0 := P2_Robot.OUT.Model45F_Vakum_ON;
	P2_Pracovisko.COM_VentilovyTerminal[0].1 := P2_Robot.OUT.Model45F_Vakum_OFF;
	P2_Pracovisko.COM_VentilovyTerminal[0].2 := P2_Robot.OUT.Model5H_Vakum_ON;
	P2_Pracovisko.COM_VentilovyTerminal[0].3 := P2_Robot.OUT.Model5H_Vakum_OFF;
	P2_Pracovisko.COM_VentilovyTerminal[0].4 := P2_Srobovanie.OUT.Skrutkovacka_M4_Prisavanie_ON;
	P2_Pracovisko.COM_VentilovyTerminal[0].5 := P2_Srobovanie.OUT.Skrutkovacka_M4_Prisavanie_OFF;
	P2_Pracovisko.COM_VentilovyTerminal[0].6 := P2_Srobovanie.OUT.Skrutkovacka_M4_Odvzdusn_ON;
	P2_Pracovisko.COM_VentilovyTerminal[0].7;

	//8-15
	P2_Pracovisko.COM_VentilovyTerminal[1].0 := P2_StoperZaklTesnenia.OUT.ZasunStoper;
	P2_Pracovisko.COM_VentilovyTerminal[1].1 := P2_StoperMaticovacky.OUT.ZasunStoper;
	P2_Pracovisko.COM_VentilovyTerminal[1].2 := P2_AkumulacnyStoper.OUT.ZasunStoper;
	P2_Pracovisko.COM_VentilovyTerminal[1].3 := P2_StoperSrobovania.OUT.ZasunStoper;
	P2_Pracovisko.COM_VentilovyTerminal[1].4 := P2_StoperZvarania.OUT.ZasunStoper;
	P2_Pracovisko.COM_VentilovyTerminal[1].5 := P2_SpodnyStoper.OUT.ZasunStoper;
	P2_Pracovisko.COM_VentilovyTerminal[1].6 := P2_Robot.OUT.ZaistiGriper;
	P2_Pracovisko.COM_VentilovyTerminal[1].7 := P2_Robot.OUT.OdistiGriper;

	//16-23
	P2_Pracovisko.COM_VentilovyTerminal[2].0 := P2_Robot.OUT.PneuZamokUchopovaca_ODOMKNI;
	P2_Pracovisko.COM_VentilovyTerminal[2].1;
	P2_Pracovisko.COM_VentilovyTerminal[2].2 := P2_StoperMaticovacky.SkrutSet_MaticaM4.OUT.ZhadzovaciVzduch_RUN;
	P2_Pracovisko.COM_VentilovyTerminal[2].3 := P2_StoperMaticovacky.SkrutSet_MaticaM4.OUT.TriediaciVzduch_RUN;
	P2_Pracovisko.COM_VentilovyTerminal[2].4 := P2_StoperMaticovacky.SkrutSet_MaticaM4.OUT.OtocOddelovacMatice_NaVystup;
	P2_Pracovisko.COM_VentilovyTerminal[2].5;
	P2_Pracovisko.COM_VentilovyTerminal[2].6 := P2_StoperMaticovacky.SkrutSet_MaticaM4.OUT.NastrelenieMatice_RUN;
	P2_Pracovisko.COM_VentilovyTerminal[2].7;

	//24-31
	P2_Pracovisko.COM_VentilovyTerminal[3].0 := P2_StoperMaticovacky.SkrutSet_MaticaM4.OUT.PodavacMatice_Vysun;
	P2_Pracovisko.COM_VentilovyTerminal[3].1;
	P2_Pracovisko.COM_VentilovyTerminal[3].2 := P2_StoperMaticovacky.OUT.Maticovacka_M4_Prisavanie_ON;
	P2_Pracovisko.COM_VentilovyTerminal[3].3 := P2_StoperMaticovacky.OUT.Maticovacka_M4_Odvzdusn_ON;
	P2_Pracovisko.COM_VentilovyTerminal[3].4 := P2_Srobovanie.SkrutSet_M5.OUT.VibracnyHrniec.PrerusenieZasobovaniaSkrutiek;
	P2_Pracovisko.COM_VentilovyTerminal[3].5 := P2_Srobovanie.SkrutSet_M5.OUT.VibracnyHrniec.TiedenieSkrutiek;
	P2_Pracovisko.COM_VentilovyTerminal[3].6 := P2_Srobovanie.SkrutSet_M5.OUT.VibracnyHrniec.OddelovacVysunut;
	P2_Pracovisko.COM_VentilovyTerminal[3].7;

	//32-39
	P2_Pracovisko.COM_VentilovyTerminal[4].0 := P2_Srobovanie.SkrutSet_M5.OUT.VibracnyHrniec.VzduchNastreleniaSkrutky;
	P2_Pracovisko.COM_VentilovyTerminal[4].1;
	P2_Pracovisko.COM_VentilovyTerminal[4].2 := P2_Srobovanie.SkrutSet_M6.OUT.VibracnyHrniec.TiedenieSkrutiek;
	P2_Pracovisko.COM_VentilovyTerminal[4].3 := P2_Srobovanie.SkrutSet_M6.OUT.VibracnyHrniec.PrerusenieZasobovaniaSkrutiek;
	P2_Pracovisko.COM_VentilovyTerminal[4].4 := P2_Srobovanie.SkrutSet_M6.OUT.VibracnyHrniec.OddelovacVysunut;
	P2_Pracovisko.COM_VentilovyTerminal[4].5;
	P2_Pracovisko.COM_VentilovyTerminal[4].6 := P2_Srobovanie.SkrutSet_M6.OUT.VibracnyHrniec.VzduchNastreleniaSkrutky;
	P2_Pracovisko.COM_VentilovyTerminal[4].7;

	//40-47
	P2_Pracovisko.COM_VentilovyTerminal[5].0 := P2_Srobovanie.SkrutSet_M4.OUT.ZhadzovaciVzduch_RUN;
	P2_Pracovisko.COM_VentilovyTerminal[5].1 := P2_Srobovanie.SkrutSet_M4.OUT.TriediaciVzduch_RUN;
	P2_Pracovisko.COM_VentilovyTerminal[5].2 := P2_Srobovanie.SkrutSet_M4.OUT.OtocPodavac_NaVystup;
	P2_Pracovisko.COM_VentilovyTerminal[5].3 := P2_Srobovanie.SkrutSet_M4.OUT.OtocPodavac_NaVstup;
	P2_Pracovisko.COM_VentilovyTerminal[5].4 := P2_Srobovanie.OUT.Skrutkovacka_M6_Prisavanie_ON;
	P2_Pracovisko.COM_VentilovyTerminal[5].5 := P2_Srobovanie.OUT.Skrutkovacka_M6_Odvzdusn_ON;
	P2_Pracovisko.COM_VentilovyTerminal[5].6 := P2_Srobovanie.SkrutSet_M6.OUT.Brzda.PodajSkrutku;
	P2_Pracovisko.COM_VentilovyTerminal[5].7 := P2_Srobovanie.SkrutSet_M6.OUT.Brzda.ZakladnaPoloha;

	//48-55
	P2_Pracovisko.COM_VentilovyTerminal[6].0 := P2_Srobovanie.SkrutSet_M6.OUT.Brzda.OdsavanieNecistot;
	P2_Pracovisko.COM_VentilovyTerminal[6].1 := P2_Srobovanie.SkrutSet_M6.OUT.Brzda.NastrelenieSkrutky;
	P2_Pracovisko.COM_VentilovyTerminal[6].2 := P2_Srobovanie.OUT.Skrutkovacka_M5_Prisavanie_ON;
	P2_Pracovisko.COM_VentilovyTerminal[6].3 := P2_Srobovanie.OUT.Skrutkovacka_M5_Odvzdusn_ON;
	P2_Pracovisko.COM_VentilovyTerminal[6].4 := P2_Srobovanie.SkrutSet_M5.OUT.Brzda.PodajSkrutku;
	P2_Pracovisko.COM_VentilovyTerminal[6].5 := P2_Srobovanie.SkrutSet_M5.OUT.Brzda.ZakladnaPoloha;
	P2_Pracovisko.COM_VentilovyTerminal[6].6 := P2_Srobovanie.SkrutSet_M5.OUT.Brzda.OdsavanieNecistot;
	P2_Pracovisko.COM_VentilovyTerminal[6].7 := P2_Srobovanie.SkrutSet_M5.OUT.Brzda.NastrelenieSkrutky;

	//56-63
	P2_Pracovisko.COM_VentilovyTerminal[7].0 := P2_Cistenie.OUT.VzduchPreIonizator_ON;
	P2_Pracovisko.COM_VentilovyTerminal[7].1 := P2_Cistenie.OUT.OdsavanieOfuk_ON;
	P2_Pracovisko.COM_VentilovyTerminal[7].2 := P2_Cistenie.OUT.Odsavanie_ON;
	P2_Pracovisko.COM_VentilovyTerminal[7].3;
	P2_Pracovisko.COM_VentilovyTerminal[7].4;
	P2_Pracovisko.COM_VentilovyTerminal[7].5;
	P2_Pracovisko.COM_VentilovyTerminal[7].6;
	P2_Pracovisko.COM_VentilovyTerminal[7].7;

	//64-71
	P2_Pracovisko.COM_VentilovyTerminal[8].0;
	P2_Pracovisko.COM_VentilovyTerminal[8].1:= P2_StoperMaticovacky.OUT.Maticovacka_M4_Pneuzamok_ODOMKNI;
	P2_Pracovisko.COM_VentilovyTerminal[8].2;
	P2_Pracovisko.COM_VentilovyTerminal[8].3;
	P2_Pracovisko.COM_VentilovyTerminal[8].4 := P2_StoperMaticovacky.OUT.Maticovacku_M4_VYSUN;
	P2_Pracovisko.COM_VentilovyTerminal[8].5;
	P2_Pracovisko.COM_VentilovyTerminal[8].6 := P2_StoperMaticovacky.OUT.Centrovanie_VYSUN;
	P2_Pracovisko.COM_VentilovyTerminal[8].7 := P2_StoperMaticovacky.OUT.Centrovanie_ZASUN;

	//72-79
	P2_Pracovisko.COM_VentilovyTerminal[9].0 := P2_StoperSrobovania.OUT.Centrovanie_VYSUN;
	P2_Pracovisko.COM_VentilovyTerminal[9].1 := P2_StoperSrobovania.OUT.Centrovanie_ZASUN;
	P2_Pracovisko.COM_VentilovyTerminal[9].2 := P2_StoperZvarania.OUT.Centrovanie_VYSUN;
	P2_Pracovisko.COM_VentilovyTerminal[9].3 := P2_StoperZvarania.OUT.Centrovanie_ZASUN;
	P2_Pracovisko.COM_VentilovyTerminal[9].4;
	P2_Pracovisko.COM_VentilovyTerminal[9].5;
	P2_Pracovisko.COM_VentilovyTerminal[9].6 := P2_Srobovanie.OUT.Skrutkovacku_M6_VYSUN;
	P2_Pracovisko.COM_VentilovyTerminal[9].7;

	IF NOT P2_Robot.OUT.PneuZamokUchopovaca_ODOMKNI THEN
		P2_Pracovisko.COM_VentilovyTerminal[9].4 := FALSE;
		P2_Pracovisko.COM_VentilovyTerminal[9].5 := FALSE;
	ELSIF P2_Robot.OUT.Griper_OTVOR THEN
		P2_Pracovisko.COM_VentilovyTerminal[9].4 := TRUE;
		P2_Pracovisko.COM_VentilovyTerminal[9].5 := FALSE;
	ELSIF P2_Robot.OUT.Griper_ZATVOR THEN
		P2_Pracovisko.COM_VentilovyTerminal[9].4 := FALSE;
		P2_Pracovisko.COM_VentilovyTerminal[9].5 := TRUE;
	END_IF

	//80-87
	P2_Pracovisko.COM_VentilovyTerminal[10].0 := P2_Srobovanie.OUT.Skrutkovacku_M5_VYSUN;
	P2_Pracovisko.COM_VentilovyTerminal[10].1;
	P2_Pracovisko.COM_VentilovyTerminal[10].2 := P2_Zvaranie.OUT.PresunZvarania_VLAVO;
	P2_Pracovisko.COM_VentilovyTerminal[10].3 := P2_Zvaranie.OUT.PresunZvaranie_VPRAVO;
	P2_Pracovisko.COM_VentilovyTerminal[10].4 := P2_Cistenie.OUT.Dvere_OTVOR;
	P2_Pracovisko.COM_VentilovyTerminal[10].5 := P2_Cistenie.OUT.Dvere_ZATVOR;
	P2_Pracovisko.COM_VentilovyTerminal[10].6;
	P2_Pracovisko.COM_VentilovyTerminal[10].7;

	//Volanie knižnic//
	P2_ZakladacTesnenia.ServoPojazduZakladaca();
	P2_ZakladacTesnenia.ServoZdvihuZakladaca();
	P2_StoperMaticovacky.SkrutSet_MaticaM4();
	P2_Srobovanie.SkrutSet_M4();
	P2_Srobovanie.SkrutSet_M5();
	P2_Srobovanie.SkrutSet_M6();
	P2_Srobovanie.ServoManipulOsX();
	P2_Srobovanie.ServoManipulOsY();
	P2_Srobovanie.ServoManipulOsZ_M4();
	P2_Zvaranie.ServoZdvihuZvarania();

END_PROGRAM

PROGRAM _EXIT
	(* Insert code here *)

END_PROGRAM
```

#### Variables.var - Local variables
```iecst
VAR
	Convert_0 : UsintToUint := (0);
	Convert_1 : UsintToUint := (0);
	Convert_2 : UsintToUint := (0);
	Convert_3 : UsintToUint := (0);
END_VAR
```

### Program Logical/Program/Pracovisko_3/P3_Main (IEC)

#### Main.st - Init, cyclic, exit code
```iecst
PROGRAM _INIT
	(* Insert code here *)

END_PROGRAM

PROGRAM _CYCLIC

	//Volanie podprogramov//
	ProfinetKomunikaciaKAM13;

	//Odomknutie pneumatického zámku zdvižiek//
	IF Safety.STAV.P3_ZonaBunky_AKTIVNA THEN
		P3_Pracovisko.OUT.ZdvizkyPneuZamok_ODOMKNI:= TRUE;
	ELSE
		P3_Pracovisko.OUT.ZdvizkyPneuZamok_ODOMKNI:= FALSE;
	END_IF

	//**************************************Ukončenie cyklu pracoviska****************************************************//
	IF P3_Pracovisko.KoniecCyklu THEN
		IF P3_Dopravniky.Automat THEN
			P3_Dopravniky.KoniecCyklu:= TRUE;
		END_IF
		IF P3_SpodnyStoper.Automat THEN
			P3_SpodnyStoper.KoniecCyklu:= TRUE;
		END_IF
		IF P3_StoperSrobovania.Automat THEN
			P3_StoperSrobovania.KoniecCyklu:= TRUE;
		END_IF
		IF P3_Srobovanie.Automat THEN
			P3_Srobovanie.KoniecCyklu:= TRUE;
		END_IF
		IF P3_HV_Test.Automat THEN
			P3_HV_Test.KoniecCyklu:= TRUE;
		END_IF
		IF P3_ZdvizkaPredLeakTestA.Automat THEN
			P3_ZdvizkaPredLeakTestA.KoniecCyklu:= TRUE;
		END_IF
		IF P3_ZdvizkaPredLeakTestB.Automat THEN
			P3_ZdvizkaPredLeakTestB.KoniecCyklu:= TRUE;
		END_IF
		IF P3_LeakageTestA.Automat THEN
			P3_LeakageTestA.KoniecCyklu:= TRUE;
		END_IF
		IF P3_LeakageTestB.Automat THEN
			P3_LeakageTestB.KoniecCyklu:= TRUE;
		END_IF
		IF P3_ZdvizkaZaLeakTestA.Automat THEN
			P3_ZdvizkaZaLeakTestA.KoniecCyklu:= TRUE;
		END_IF
		IF P3_ZdvizkaZaLeakTestB.Automat THEN
			P3_ZdvizkaZaLeakTestB.KoniecCyklu:= TRUE;
		END_IF
		P3_Pracovisko.KoniecCyklu:= FALSE;
	END_IF

	//************************************Ukončenie cyklu pri poruche*****************************************//
	//ST1 - Šrobovanie//
	IF P3_Pracovisko.STAV.Porucha_ST1 THEN
		IF P3_Dopravniky.Automat THEN
			P3_Dopravniky.KoniecCyklu:= TRUE;
		END_IF
		IF P3_SpodnyStoper.Automat THEN
			P3_SpodnyStoper.KoniecCyklu:= TRUE;
		END_IF
		IF P3_Srobovanie.Automat THEN
			P3_Srobovanie.Reset:= TRUE;
		END_IF
		IF P3_HV_Test.Automat THEN
			P3_HV_Test.KoniecCyklu:= TRUE;
		END_IF
		IF P3_ZdvizkaPredLeakTestA.Automat THEN
			P3_ZdvizkaPredLeakTestA.KoniecCyklu:= TRUE;
		END_IF
		IF P3_ZdvizkaPredLeakTestB.Automat THEN
			P3_ZdvizkaPredLeakTestB.KoniecCyklu:= TRUE;
		END_IF
		IF P3_LeakageTestA.Automat THEN
			P3_LeakageTestA.KoniecCyklu:= TRUE;
		END_IF
		IF P3_LeakageTestB.Automat THEN
			P3_LeakageTestB.KoniecCyklu:= TRUE;
		END_IF
		IF P3_ZdvizkaZaLeakTestA.Automat THEN
			P3_ZdvizkaZaLeakTestA.KoniecCyklu:= TRUE;
		END_IF
		IF P3_ZdvizkaZaLeakTestB.Automat THEN
			P3_ZdvizkaZaLeakTestB.KoniecCyklu:= TRUE;
		END_IF
	END_IF

	//ST2 - HV test//
	IF P3_Pracovisko.STAV.Porucha_ST2 THEN
		IF P3_Dopravniky.Automat THEN
			P3_Dopravniky.KoniecCyklu:= TRUE;
		END_IF
		IF P3_SpodnyStoper.Automat THEN
			P3_SpodnyStoper.KoniecCyklu:= TRUE;
		END_IF
		IF P3_StoperSrobovania.Automat THEN
			P3_StoperSrobovania.KoniecCyklu:= TRUE;
		END_IF
		IF P3_Srobovanie.Automat THEN
			P3_Srobovanie.KoniecCyklu:= TRUE;
		END_IF
		IF P3_HV_Test.Automat THEN
			P3_HV_Test.Reset:= TRUE;
		END_IF
		IF P3_ZdvizkaPredLeakTestA.Automat THEN
			P3_ZdvizkaPredLeakTestA.KoniecCyklu:= TRUE;
		END_IF
		IF P3_ZdvizkaPredLeakTestB.Automat THEN
			P3_ZdvizkaPredLeakTestB.KoniecCyklu:= TRUE;
		END_IF
		IF P3_LeakageTestA.Automat THEN
			P3_LeakageTestA.KoniecCyklu:= TRUE;
		END_IF
		IF P3_LeakageTestB.Automat THEN
			P3_LeakageTestB.KoniecCyklu:= TRUE;
		END_IF
		IF P3_ZdvizkaZaLeakTestA.Automat THEN
			P3_ZdvizkaZaLeakTestA.KoniecCyklu:= TRUE;
		END_IF
		IF P3_ZdvizkaZaLeakTestB.Automat THEN
			P3_ZdvizkaZaLeakTestB.KoniecCyklu:= TRUE;
		END_IF
	END_IF

	//ST3 - Zdvižka pred Leakage testom A//
	IF P3_Pracovisko.STAV.Porucha_ST3 THEN
		IF P3_Dopravniky.Automat THEN
			P3_Dopravniky.KoniecCyklu:= TRUE;
		END_IF
		IF P3_SpodnyStoper.Automat THEN
			P3_SpodnyStoper.KoniecCyklu:= TRUE;
		END_IF
		IF P3_StoperSrobovania.Automat THEN
			P3_StoperSrobovania.KoniecCyklu:= TRUE;
		END_IF
		IF P3_Srobovanie.Automat THEN
			P3_Srobovanie.KoniecCyklu:= TRUE;
		END_IF
		IF P3_HV_Test.Automat THEN
			P3_HV_Test.KoniecCyklu:= TRUE;
		END_IF
		IF P3_ZdvizkaPredLeakTestA.Automat THEN
			P3_ZdvizkaPredLeakTestA.Reset:= TRUE;
		END_IF
		IF P3_ZdvizkaPredLeakTestB.Automat THEN
			P3_ZdvizkaPredLeakTestB.KoniecCyklu:= TRUE;
		END_IF
		IF P3_LeakageTestA.Automat THEN
			P3_LeakageTestA.KoniecCyklu:= TRUE;
		END_IF
		IF P3_LeakageTestB.Automat THEN
			P3_LeakageTestB.KoniecCyklu:= TRUE;
		END_IF
		IF P3_ZdvizkaZaLeakTestA.Automat THEN
			P3_ZdvizkaZaLeakTestA.KoniecCyklu:= TRUE;
		END_IF
		IF P3_ZdvizkaZaLeakTestB.Automat THEN
			P3_ZdvizkaZaLeakTestB.KoniecCyklu:= TRUE;
		END_IF
	END_IF

	//ST4 - Zdvižka pred Leakage testom B//
	IF P3_Pracovisko.STAV.Porucha_ST4 THEN
		IF P3_Dopravniky.Automat THEN
			P3_Dopravniky.KoniecCyklu:= TRUE;
		END_IF
		IF P3_SpodnyStoper.Automat THEN
			P3_SpodnyStoper.KoniecCyklu:= TRUE;
		END_IF
		IF P3_StoperSrobovania.Automat THEN
			P3_StoperSrobovania.KoniecCyklu:= TRUE;
		END_IF
		IF P3_Srobovanie.Automat THEN
			P3_Srobovanie.KoniecCyklu:= TRUE;
		END_IF
		IF P3_HV_Test.Automat THEN
			P3_HV_Test.KoniecCyklu:= TRUE;
		END_IF
		IF P3_ZdvizkaPredLeakTestA.Automat THEN
			P3_ZdvizkaPredLeakTestA.KoniecCyklu:= TRUE;
		END_IF
		IF P3_ZdvizkaPredLeakTestB.Automat THEN
			P3_ZdvizkaPredLeakTestB.Reset:= TRUE;
		END_IF
		IF P3_LeakageTestA.Automat THEN
			P3_LeakageTestA.KoniecCyklu:= TRUE;
		END_IF
		IF P3_LeakageTestB.Automat THEN
			P3_LeakageTestB.KoniecCyklu:= TRUE;
		END_IF
		IF P3_ZdvizkaZaLeakTestA.Automat THEN
			P3_ZdvizkaZaLeakTestA.KoniecCyklu:= TRUE;
		END_IF
		IF P3_ZdvizkaZaLeakTestB.Automat THEN
			P3_ZdvizkaZaLeakTestB.KoniecCyklu:= TRUE;
		END_IF
	END_IF

	//ST5 - Leakage test A//
	IF P3_Pracovisko.STAV.Porucha_ST5 THEN
		IF P3_Dopravniky.Automat THEN
			P3_Dopravniky.KoniecCyklu:= TRUE;
		END_IF
		IF P3_SpodnyStoper.Automat THEN
			P3_SpodnyStoper.KoniecCyklu:= TRUE;
		END_IF
		IF P3_StoperSrobovania.Automat THEN
			P3_StoperSrobovania.KoniecCyklu:= TRUE;
		END_IF
		IF P3_Srobovanie.Automat THEN
			P3_Srobovanie.KoniecCyklu:= TRUE;
		END_IF
		IF P3_HV_Test.Automat THEN
			P3_HV_Test.KoniecCyklu:= TRUE;
		END_IF
		IF P3_ZdvizkaPredLeakTestA.Automat THEN
			P3_ZdvizkaPredLeakTestA.KoniecCyklu:= TRUE;
		END_IF
		IF P3_ZdvizkaPredLeakTestB.Automat THEN
			P3_ZdvizkaPredLeakTestB.KoniecCyklu:= TRUE;
		END_IF
		IF P3_LeakageTestA.Automat THEN
			P3_LeakageTestA.Reset:= TRUE;
		END_IF
		IF P3_LeakageTestB.Automat THEN
			P3_LeakageTestB.KoniecCyklu:= TRUE;
		END_IF
		IF P3_ZdvizkaZaLeakTestA.Automat THEN
			P3_ZdvizkaZaLeakTestA.KoniecCyklu:= TRUE;
		END_IF
		IF P3_ZdvizkaZaLeakTestB.Automat THEN
			P3_ZdvizkaZaLeakTestB.KoniecCyklu:= TRUE;
		END_IF
	END_IF

	//ST6 - Leakage test B//
	IF P3_Pracovisko.STAV.Porucha_ST6 THEN
		IF P3_Dopravniky.Automat THEN
			P3_Dopravniky.KoniecCyklu:= TRUE;
		END_IF
		IF P3_SpodnyStoper.Automat THEN
			P3_SpodnyStoper.KoniecCyklu:= TRUE;
		END_IF
		IF P3_StoperSrobovania.Automat THEN
			P3_StoperSrobovania.KoniecCyklu:= TRUE;
		END_IF
		IF P3_Srobovanie.Automat THEN
			P3_Srobovanie.KoniecCyklu:= TRUE;
		END_IF
		IF P3_HV_Test.Automat THEN
			P3_HV_Test.KoniecCyklu:= TRUE;
		END_IF
		IF P3_ZdvizkaPredLeakTestA.Automat THEN
			P3_ZdvizkaPredLeakTestA.KoniecCyklu:= TRUE;
		END_IF
		IF P3_ZdvizkaPredLeakTestB.Automat THEN
			P3_ZdvizkaPredLeakTestB.KoniecCyklu:= TRUE;
		END_IF
		IF P3_LeakageTestA.Automat THEN
			P3_LeakageTestA.KoniecCyklu:= TRUE;
		END_IF
		IF P3_LeakageTestB.Automat THEN
			P3_LeakageTestB.Reset:= TRUE;
		END_IF
		IF P3_ZdvizkaZaLeakTestA.Automat THEN
			P3_ZdvizkaZaLeakTestA.KoniecCyklu:= TRUE;
		END_IF
		IF P3_ZdvizkaZaLeakTestB.Automat THEN
			P3_ZdvizkaZaLeakTestB.KoniecCyklu:= TRUE;
		END_IF
	END_IF

	//ST7 - Zdvižka za Leakage testom A//
	IF P3_Pracovisko.STAV.Porucha_ST7 THEN
		IF P3_Dopravniky.Automat THEN
			P3_Dopravniky.KoniecCyklu:= TRUE;
		END_IF
		IF P3_SpodnyStoper.Automat THEN
			P3_SpodnyStoper.KoniecCyklu:= TRUE;
		END_IF
		IF P3_StoperSrobovania.Automat THEN
			P3_StoperSrobovania.KoniecCyklu:= TRUE;
		END_IF
		IF P3_Srobovanie.Automat THEN
			P3_Srobovanie.KoniecCyklu:= TRUE;
		END_IF
		IF P3_HV_Test.Automat THEN
			P3_HV_Test.KoniecCyklu:= TRUE;
		END_IF
		IF P3_ZdvizkaPredLeakTestA.Automat THEN
			P3_ZdvizkaPredLeakTestA.KoniecCyklu:= TRUE;
		END_IF
		IF P3_ZdvizkaPredLeakTestB.Automat THEN
			P3_ZdvizkaPredLeakTestB.KoniecCyklu:= TRUE;
		END_IF
		IF P3_LeakageTestA.Automat THEN
			P3_LeakageTestA.KoniecCyklu:= TRUE;
		END_IF
		IF P3_LeakageTestB.Automat THEN
			P3_LeakageTestB.KoniecCyklu:= TRUE;
		END_IF
		IF P3_ZdvizkaZaLeakTestA.Automat THEN
			P3_ZdvizkaZaLeakTestA.Reset:= TRUE;
		END_IF
		IF P3_ZdvizkaZaLeakTestB.Automat THEN
			P3_ZdvizkaZaLeakTestB.KoniecCyklu:= TRUE;
		END_IF
	END_IF

	//ST8 - Zdvižka za Leakage testom B//
	IF P3_Pracovisko.STAV.Porucha_ST8 THEN
		IF P3_Dopravniky.Automat THEN
			P3_Dopravniky.KoniecCyklu:= TRUE;
		END_IF
		IF P3_SpodnyStoper.Automat THEN
			P3_SpodnyStoper.KoniecCyklu:= TRUE;
		END_IF
		IF P3_StoperSrobovania.Automat THEN
			P3_StoperSrobovania.KoniecCyklu:= TRUE;
		END_IF
		IF P3_Srobovanie.Automat THEN
			P3_Srobovanie.KoniecCyklu:= TRUE;
		END_IF
		IF P3_HV_Test.Automat THEN
			P3_HV_Test.KoniecCyklu:= TRUE;
		END_IF
		IF P3_ZdvizkaPredLeakTestA.Automat THEN
			P3_ZdvizkaPredLeakTestA.KoniecCyklu:= TRUE;
		END_IF
		IF P3_ZdvizkaPredLeakTestB.Automat THEN
			P3_ZdvizkaPredLeakTestB.KoniecCyklu:= TRUE;
		END_IF
		IF P3_LeakageTestA.Automat THEN
			P3_LeakageTestA.KoniecCyklu:= TRUE;
		END_IF
		IF P3_LeakageTestB.Automat THEN
			P3_LeakageTestB.KoniecCyklu:= TRUE;
		END_IF
		IF P3_ZdvizkaZaLeakTestA.Automat THEN
			P3_ZdvizkaZaLeakTestA.KoniecCyklu:= TRUE;
		END_IF
		IF P3_ZdvizkaZaLeakTestB.Automat THEN
			P3_ZdvizkaZaLeakTestB.Reset:= TRUE;
		END_IF
	END_IF

	//*********************************Status prebieha ukončenie cyklu********************************************//
	IF P3_Dopravniky.KoniecCyklu OR
		P3_SpodnyStoper.KoniecCyklu OR
		P3_StoperSrobovania.KoniecCyklu OR
		P3_Srobovanie.KoniecCyklu OR
		P3_HV_Test.KoniecCyklu OR
		P3_ZdvizkaPredLeakTestA.KoniecCyklu OR
		P3_ZdvizkaPredLeakTestB.KoniecCyklu OR
		P3_LeakageTestA.KoniecCyklu OR
		P3_LeakageTestB.KoniecCyklu OR
		P3_ZdvizkaZaLeakTestA.KoniecCyklu OR
		P3_ZdvizkaZaLeakTestB.KoniecCyklu THEN
		P3_Pracovisko.STAV.UkoncenieCyklu_BUSY:= TRUE;
	ELSE
		P3_Pracovisko.STAV.UkoncenieCyklu_BUSY:= FALSE;
	END_IF

	//******************************************Resetovanie pracoviska************************************************************//
	IF P3_Pracovisko.Reset THEN
		P3_Dopravniky.Reset:= TRUE;
		P3_SpodnyStoper.Reset:= TRUE;
		P3_StoperSrobovania.Reset:= TRUE;
		P3_Srobovanie.Reset:= TRUE;
		P3_HV_Test.Reset:= TRUE;
		P3_ZdvizkaPredLeakTestA.Reset:= TRUE;
		P3_ZdvizkaPredLeakTestB.Reset:= TRUE;
		P3_LeakageTestA.Reset:= TRUE;
		P3_LeakageTestB.Reset:= TRUE;
		P3_ZdvizkaZaLeakTestA.Reset:= TRUE;
		P3_ZdvizkaZaLeakTestB.Reset:= TRUE;
		P3_Pracovisko.STAV.Porucha_ST1:= FALSE;
		P3_Pracovisko.STAV.Porucha_ST2:= FALSE;
		P3_Pracovisko.STAV.Porucha_ST3:= FALSE;
		P3_Pracovisko.STAV.Porucha_ST4:= FALSE;
		P3_Pracovisko.STAV.Porucha_ST5:= FALSE;
		P3_Pracovisko.STAV.Porucha_ST6:= FALSE;
		P3_Pracovisko.STAV.Porucha_ST7:= FALSE;
		P3_Pracovisko.STAV.Porucha_ST8:= FALSE;
		P3_Pracovisko.Reset:= FALSE;
	END_IF

	//Prepnutie pracoviska do manualneho režimu//
	IF P3_Pracovisko.Manual THEN
		P3_Dopravniky.Manual:= TRUE;
		P3_SpodnyStoper.Manual:= TRUE;
		P3_StoperSrobovania.Manual:= TRUE;
		P3_Srobovanie.Manual:= TRUE;
		P3_HV_Test.Manual:= TRUE;
		P3_ZdvizkaPredLeakTestA.Manual:= TRUE;
		P3_ZdvizkaPredLeakTestB.Manual:= TRUE;
		P3_LeakageTestA.Manual:= TRUE;
		P3_LeakageTestB.Manual:= TRUE;
		P3_ZdvizkaZaLeakTestA.Manual:= TRUE;
		P3_ZdvizkaZaLeakTestB.Manual:= TRUE;
		P3_Pracovisko.Manual:= FALSE;
	END_IF

	//Spustenie pracoviska v automatickom režime//
	IF P3_Pracovisko.Automat THEN
		IF Safety.STAV.P3_ZonaBunky_AKTIVNA AND P3_Pracovisko.STAV.HardwareBunky_OK THEN
			P3_Dopravniky.Automat:= TRUE;
			P3_SpodnyStoper.Automat:= TRUE;
			P3_StoperSrobovania.Automat:= TRUE;
			P3_Srobovanie.Automat:= TRUE;
			P3_HV_Test.Automat:= TRUE;
			P3_ZdvizkaPredLeakTestA.Automat:= TRUE;
			P3_ZdvizkaPredLeakTestB.Automat:= TRUE;
			P3_LeakageTestA.Automat:= TRUE;
			P3_LeakageTestB.Automat:= TRUE;
			P3_ZdvizkaZaLeakTestA.Automat:= TRUE;
			P3_ZdvizkaZaLeakTestB.Automat:= TRUE;
		END_IF
		P3_Pracovisko.Automat:= FALSE;
	END_IF

	//***************************************************Príznaky pracoviska******************************************************//
	//Príznak pracovisko stav AUTOMAT//
	IF P3_Dopravniky.Automat OR
		P3_SpodnyStoper.Automat OR
		P3_StoperSrobovania.Automat OR
		P3_Srobovanie.Automat OR
		P3_HV_Test.Automat OR
		P3_ZdvizkaPredLeakTestA.Automat OR
		P3_ZdvizkaPredLeakTestB.Automat OR
		P3_LeakageTestA.Automat OR
		P3_LeakageTestB.Automat OR
		P3_ZdvizkaZaLeakTestA.Automat OR
		P3_ZdvizkaZaLeakTestB.Automat THEN
		P3_Pracovisko.STAV.Automat:= TRUE;
	ELSE
		P3_Pracovisko.STAV.Automat:= FALSE;
	END_IF

	//Priznak pracovisko stav MANUAL//
	IF P3_Dopravniky.Manual OR
		P3_SpodnyStoper.Manual OR
		P3_StoperSrobovania.Manual OR
		P3_Srobovanie.Manual OR
		P3_HV_Test.Manual OR
		P3_ZdvizkaPredLeakTestA.Manual OR
		P3_ZdvizkaPredLeakTestB.Manual OR
		P3_LeakageTestA.Manual OR
		P3_LeakageTestB.Manual OR
		P3_ZdvizkaZaLeakTestA.Manual OR
		P3_ZdvizkaZaLeakTestB.Manual THEN
		P3_Pracovisko.STAV.Manual:= TRUE;
	ELSE
		P3_Pracovisko.STAV.Manual:= FALSE;
	END_IF

	//Príznak pracovisko stav PoINIT//
	IF P3_Dopravniky.STAV.PoINIT AND
		P3_SpodnyStoper.STAV.PoINIT AND
		P3_StoperSrobovania.STAV.PoINIT AND
		P3_Srobovanie.STAV.PoINIT AND
		P3_HV_Test.STAV.PoINIT AND
		P3_ZdvizkaPredLeakTestA.STAV.PoINIT AND
		P3_ZdvizkaPredLeakTestB.STAV.PoINIT AND
		P3_LeakageTestA.STAV.PoINIT AND
		P3_LeakageTestB.STAV.PoINIT AND
		P3_ZdvizkaZaLeakTestA.STAV.PoINIT AND
		P3_ZdvizkaZaLeakTestB.STAV.PoINIT THEN
		P3_Pracovisko.STAV.PoINIT:= TRUE;
	ELSE
		P3_Pracovisko.STAV.PoINIT:= FALSE;
	END_IF

	//Príznak pracovisko stav READY//
	IF SC_P3_Dopravniky.Step = 1 AND
		SC_P3_SpodnyStoper.Step = 1 AND
		SC_P3_StoperSrobovania.Step = 1 AND
		SC_P3_Srobovanie.Step = 1 AND
		SC_P3_HV_Test.Step = 1 AND
		SC_P3_ZdvizkaPredLeakTestA.Step = 1 AND
		SC_P3_ZdvizkaPredLeakTestB.Step = 1 AND
		SC_P3_LeakageTestA.Step = 1 AND
		SC_P3_LeakageTestB.Step = 1 AND
		SC_P3_ZdvizkaZaLeakTestA.Step = 1 AND
		SC_P3_ZdvizkaZaLeakTestB.Step = 1 THEN
		P3_Pracovisko.STAV.READY:= TRUE;
	ELSE
		P3_Pracovisko.STAV.READY:= FALSE;
	END_IF

	//Príznak pracovisko stav PORUCHA//
	IF P3_Pracovisko.STAV.Porucha_ST1 OR
		P3_Pracovisko.STAV.Porucha_ST2 OR
		P3_Pracovisko.STAV.Porucha_ST3 OR
		P3_Pracovisko.STAV.Porucha_ST4 OR
		P3_Pracovisko.STAV.Porucha_ST5 OR
		P3_Pracovisko.STAV.Porucha_ST6 OR
		P3_Pracovisko.STAV.Porucha_ST7 OR
		P3_Pracovisko.STAV.Porucha_ST8 THEN
		P3_Pracovisko.STAV.PORUCHA:= TRUE;
	ELSE
		P3_Pracovisko.STAV.PORUCHA:= FALSE;
	END_IF

	//Príznak HW Bunky OK//
	IF P3_Pracovisko.IN.TlakVzduchu_OK AND
		P3_Pracovisko.IN.ModulFesto_IO_KomOK AND
		P3_Pracovisko.IN.ModulWeidmuller_IO_KomOK AND
		(*P3_Pracovisko.IN.Kamery_ControlUnit_KomOK AND*)
		P3_Pracovisko.IN.LeakageTesterA_KomOK AND
		P3_Pracovisko.IN.LeakageTesterB_KomOK AND
		P3_Pracovisko.IN.ServoManipulatorOsY_KomOK AND
		P3_Pracovisko.IN.ServoManipulatorOsZ_M5_KomOK AND
		P3_Pracovisko.IN.Skrutkovacka_K40_KomOK AND
		P3_Pracovisko.IN.Skrutkovacka_M5_KomOK AND
		P3_Srobovanie.IN.NapajanieSkrutkovackyK40_OK AND
		P3_Srobovanie.IN.NapajanieSkrutkovackyM5_OK AND
		P3_Srobovanie.IN.NapajanieVibrolistyM5_OK AND
		P3_Srobovanie.IN.NapajanieZasobnikaK40_OK AND
		P3_Srobovanie.IN.NapajanieZasobnikaM5_OK AND
		P3_Pracovisko.IN.VentilovyTerminal_KomOK THEN
		P3_Pracovisko.STAV.HardwareBunky_OK:= TRUE;
	ELSE
		P3_Pracovisko.STAV.HardwareBunky_OK:= FALSE;
	END_IF

	//Príznak skrutkovačky zasunuté//
	IF P3_Srobovanie.IN.Skrutkovacka_K40_ZASUNUTA AND P3_Srobovanie.PAR.ManipulOsZ_M5_AktualnaPozicia < 5 THEN
		P3_Pracovisko.STAV.SkrutkovackyZasunute:= TRUE;
	ELSE
		P3_Pracovisko.STAV.SkrutkovackyZasunute:= FALSE;
	END_IF

	//Priznak HV test zasunuty//
	IF P3_HV_Test.IN.Centrovanie_ZASUNUTE AND P3_HV_Test.IN.HorneKontakty_ZASUNUTE AND P3_HV_Test.IN.SpodneKontakty_ZASUNUTE THEN
		P3_Pracovisko.STAV.HVtest_Zasunuty:= TRUE;
	ELSE
		P3_Pracovisko.STAV.HVtest_Zasunuty:= FALSE;
	END_IF

	//Priznak LeakageTest A zasunuty//
	IF P3_LeakageTestA.IN.Centrovanie_ZASUNUTE AND P3_LeakageTestA.IN.HornyPritlak_ZASUNUTY AND P3_LeakageTestA.IN.Kopito_ZASUNUTE THEN
		P3_Pracovisko.STAV.LeakageTestA_Zasunuty:= TRUE;
	ELSE
		P3_Pracovisko.STAV.LeakageTestA_Zasunuty:= FALSE;
	END_IF

	//Priznak LeakageTest B zasunuty//
	IF P3_LeakageTestB.IN.Centrovanie_ZASUNUTE AND P3_LeakageTestB.IN.HornyPritlak_ZASUNUTY AND P3_LeakageTestB.IN.Kopito_ZASUNUTE THEN
		P3_Pracovisko.STAV.LeakageTestB_Zasunuty:= TRUE;
	ELSE
		P3_Pracovisko.STAV.LeakageTestB_Zasunuty:= FALSE;
	END_IF

	//*****************************Zapnutie osvetlenia pracoviska*********************************************************//
	P3_Pracovisko.OUT.OsvetlenieBunky_ON:= TRUE;

	P3_Pracovisko.OUT.Ventilator_ON:= TRUE;

	//****************************************Ovládanie majáka***********************************************//
	//Zelené svetlo//

	IF P3_Pracovisko.STAV.Automat THEN
		P3_Pracovisko.OUT.Majak_ZeleneSvetlo_ON:= TRUE;
	ELSIF P3_Pracovisko.STAV.Manual THEN
		P3_Pracovisko.OUT.Majak_ZeleneSvetlo_ON:= Blikac500ms;
	ELSE
		P3_Pracovisko.OUT.Majak_ZeleneSvetlo_ON:= FALSE;
	END_IF

	//Oranžové svetlo//
	IF P3_Pracovisko.STAV.Automat AND NOT P3_Pracovisko.STAV.PoINIT THEN
		P3_Pracovisko.OUT.Majak_OranzoveSvetlo_ON:= TRUE;
	ELSE
		P3_Pracovisko.OUT.Majak_OranzoveSvetlo_ON:= FALSE;
	END_IF

	//Červené svetlo//
	IF NOT Safety.STAV.Linka_ZonaCS_AKTIVNA THEN
		P3_Pracovisko.OUT.Majak_CerveneSvetlo_ON:= TRUE;
	ELSIF P3_Pracovisko.STAV.Porucha_ST1 THEN
		P3_Pracovisko.OUT.Majak_CerveneSvetlo_ON:= TRUE;
	ELSIF P3_Pracovisko.STAV.Porucha_ST2 THEN
		P3_Pracovisko.OUT.Majak_CerveneSvetlo_ON:= TRUE;
	ELSIF P3_Pracovisko.STAV.Porucha_ST3 THEN
		P3_Pracovisko.OUT.Majak_CerveneSvetlo_ON:= TRUE;
	ELSIF P3_Pracovisko.STAV.Porucha_ST4 THEN
		P3_Pracovisko.OUT.Majak_CerveneSvetlo_ON:= TRUE;
	ELSIF P3_Pracovisko.STAV.Porucha_ST5 THEN
		P3_Pracovisko.OUT.Majak_CerveneSvetlo_ON:= TRUE;
	ELSIF P3_Pracovisko.STAV.Porucha_ST6 THEN
		P3_Pracovisko.OUT.Majak_CerveneSvetlo_ON:= TRUE;
	ELSIF P3_Pracovisko.STAV.Porucha_ST7 THEN
		P3_Pracovisko.OUT.Majak_CerveneSvetlo_ON:= TRUE;
	ELSIF P3_Pracovisko.STAV.Porucha_ST8 THEN
		P3_Pracovisko.OUT.Majak_CerveneSvetlo_ON:= TRUE;
	ELSE
		P3_Pracovisko.OUT.Majak_CerveneSvetlo_ON:= FALSE;
	END_IF

	//Zvuková signalizácia//
	//	IF EDGEPOS(P3_Pracovisko.STAV.Porucha_ST1) THEN
	//		P3_Pracovisko.OUT.Majak_Hukacka_ON:= Blikac500ms;
	//	ELSIF EDGEPOS(P3_Pracovisko.STAV.Porucha_ST2) THEN
	//		P3_Pracovisko.OUT.Majak_Hukacka_ON:= Blikac500ms;
	//	ELSIF EDGEPOS(P3_Pracovisko.STAV.Porucha_ST3) THEN
	//		P3_Pracovisko.OUT.Majak_Hukacka_ON:= Blikac500ms;
	//	ELSIF EDGEPOS(P3_Pracovisko.STAV.Porucha_ST4) THEN
	//		P3_Pracovisko.OUT.Majak_Hukacka_ON:= Blikac500ms;
	//	ELSIF EDGEPOS(P3_Pracovisko.STAV.Porucha_ST5) THEN
	//		P3_Pracovisko.OUT.Majak_Hukacka_ON:= Blikac500ms;
	//	ELSIF EDGEPOS(P3_Pracovisko.STAV.Porucha_ST6) THEN
	//		P3_Pracovisko.OUT.Majak_Hukacka_ON:= Blikac500ms;
	//	ELSIF EDGEPOS(P3_Pracovisko.STAV.Porucha_ST7) THEN
	//		P3_Pracovisko.OUT.Majak_Hukacka_ON:= Blikac500ms;
	//	ELSIF EDGEPOS(P3_Pracovisko.STAV.Porucha_ST8) THEN
	//		P3_Pracovisko.OUT.Majak_Hukacka_ON:= Blikac500ms;
	//	END_IF

END_PROGRAM

PROGRAM _EXIT
	(* Insert code here *)

END_PROGRAM
```

#### Variables.var - Local variables
```iecst
VAR
	Convert_0 : UsintToUint := (0);
END_VAR
```

#### ProfinetKomunikaciaKAM13.st
```iecst
ACTION ProfinetKomunikaciaKAM13:
	//Kamerová kontrola zrušená//

	//Vstupy pre kameru//
	CAM13.Profinet_PLC_OUTPUTS[0].3:= CAM13.CMD.Triger;

	//Výstupy z kamery//
	CAM13.STAV.READY:= CAM13.Profinet_PLC_INPUTS[0].0;
	CAM13.STAV.SWITCH:= CAM13.Profinet_PLC_INPUTS[0].1;
    CAM13.STAV.BUSY:= CAM13.Profinet_PLC_INPUTS[0].2;
    CAM13.STAV.Command_AKCEPTOVANY:= CAM13.Profinet_PLC_INPUTS[0].3;
    CAM13.STAV.Command_READY:= CAM13.Profinet_PLC_INPUTS[0].4;
    CAM13.STAV.Command_ERROR:= CAM13.Profinet_PLC_INPUTS[0].5;

	//Výsledky kamery//
	CAM13.RESULT.Pritomn_SkrutkyK40_TopCover_4F5F:= CAM13.Profinet_PLC_INPUTS[2].0;
	CAM13.RESULT.Pritomn_SkrutkyM5_TopCover:= CAM13.Profinet_PLC_INPUTS[2].1;

	//Stav výsledky READY//
	IF EDGE(CAM13.STAV.SWITCH)THEN
		CAM13.STAV.Results_READY:= TRUE;
	END_IF

	//Run counter kamery//
	Convert_0.IN_Byte0:= CAM13.STAV.RunCounter_Byte1;
	Convert_0.IN_Byte1:= CAM13.STAV.RunCounter_Byte0;

	CAM13.STAV.RunCounter:= Convert_0.OUT_UINT;
	Convert_0();

END_ACTION
```

### Program Logical/Program/Pracovisko_3/P3_Dopravniky (IEC)
